LIN {X 0,Y 523.911,Z 275.225,A -85,B 0,C 180,E1 -4740.684,E2 -4740.684} C_VEL
LIN {X 0,Y 523.877,Z 275.226,A -85,B 0,C 180,E1 -4743.728,E2 -4743.728} C_VEL
LIN {X 0,Y 523.895,Z 275.245,A -85,B 0,C 180,E1 -4745.635,E2 -4745.635} C_VEL
LIN {X 0,Y 525.895,Z 284.56,A -85,B 0,C 180,E1 -4746.994,E2 -4746.994} C_VEL
LIN {X 0,Y 525.585,Z 301.308,A -85,B 0,C 180,E1 -4749.228,E2 -4749.228} C_VEL
LIN {X 0,Y 524.945,Z 326.375,A -85,B 0,C 180,E1 -4752.472,E2 -4752.472} C_VEL
LIN {X 0,Y 524.516,Z 345.364,A -85,B 0,C 180,E1 -4754.915,E2 -4754.915} C_VEL
LIN {X 0,Y 525.812,Z 356.161,A -85,B 0,C 180,E1 -4755.107,E2 -4755.107} C_VEL
LIN {X 0,Y 525.364,Z 452.042,A -85,B 0,C 180,E1 -4756.44,E2 -4756.44} C_VEL
LIN {X 0,Y 525.191,Z 462.116,A -85,B 0,C 180,E1 -4756.657,E2 -4756.657} C_VEL
LIN {X 0,Y 525.048,Z 472.823,A -85,B 0,C 180,E1 -4756.998,E2 -4756.998} C_VEL
LIN {X 0,Y 524.857,Z 483.102,A -85,B 0,C 180,E1 -4757.435,E2 -4757.435} C_VEL
LIN {X 0,Y 524.646,Z 493.466,A -85,B 0,C 180,E1 -4758.001,E2 -4758.001} C_VEL
LIN {X 0,Y 524.354,Z 503.711,A -85,B 0,C 180,E1 -4758.698,E2 -4758.698} C_VEL
LIN {X 0,Y 524.185,Z 512.016,A -85,B 0,C 180,E1 -4759.379,E2 -4759.379} C_VEL
LIN {X 0,Y 523.994,Z 520.012,A -85,B 0,C 180,E1 -4760.156,E2 -4760.156} C_VEL
LIN {X 0,Y 523.81,Z 528.29,A -85,B 0,C 180,E1 -4761.126,E2 -4761.126} C_VEL
LIN {X 0,Y 523.66,Z 535.18,A -85,B 0,C 180,E1 -4762.095,E2 -4762.095} C_VEL
LIN {X 0,Y 523.509,Z 540.935,A -85,B 0,C 180,E1 -4763.063,E2 -4763.063} C_VEL
LIN {X 0,Y 523.494,Z 546.516,A -85,B 0,C 180,E1 -4764.223,E2 -4764.223} C_VEL
LIN {X 0,Y 523.362,Z 550.893,A -85,B 0,C 180,E1 -4765.381,E2 -4765.381} C_VEL
LIN {X 0,Y 523.44,Z 553.228,A -85,B 0,C 180,E1 -4766.153,E2 -4766.153} C_VEL
LIN {X 0,Y 523.331,Z 556.518,A -85,B 0,C 180,E1 -4767.693,E2 -4767.693} C_VEL
LIN {X 0,Y 523.251,Z 558.064,A -85,B 0,C 180,E1 -4769.232,E2 -4769.232} C_VEL
LIN {X 0,Y 523.253,Z 558.357,A -85,B 0,C 180,E1 -4770.002,E2 -4770.002} C_VEL
LIN {X 0,Y 523.272,Z 557.477,A -85,B 0,C 180,E1 -4771.541,E2 -4771.541} C_VEL
LIN {X 0,Y 523.332,Z 556.501,A -85,B 0,C 180,E1 -4772.31,E2 -4772.31} C_VEL
LIN {X 0,Y 523.441,Z 553.195,A -85,B 0,C 180,E1 -4773.85,E2 -4773.85} C_VEL
LIN {X 0,Y 523.387,Z 549.529,A -85,B 0,C 180,E1 -4775.008,E2 -4775.008} C_VEL
LIN {X 0,Y 523.437,Z 544.168,A -85,B 0,C 180,E1 -4776.28,E2 -4776.28} C_VEL
LIN {X 0,Y 523.593,Z 538.647,A -85,B 0,C 180,E1 -4777.327,E2 -4777.327} C_VEL
LIN {X 0,Y 523.729,Z 532.476,A -85,B 0,C 180,E1 -4778.295,E2 -4778.295} C_VEL
LIN {X 0,Y 523.867,Z 525.025,A -85,B 0,C 180,E1 -4779.265,E2 -4779.265} C_VEL
LIN {X 0,Y 524.057,Z 515.954,A -85,B 0,C 180,E1 -4780.236,E2 -4780.236} C_VEL
LIN {X 0,Y 524.311,Z 507.212,A -85,B 0,C 180,E1 -4781.012,E2 -4781.012} C_VEL
LIN {X 0,Y 524.498,Z 498.064,A -85,B 0,C 180,E1 -4781.689,E2 -4781.689} C_VEL
LIN {X 0,Y 524.739,Z 487.826,A -85,B 0,C 180,E1 -4782.306,E2 -4782.306} C_VEL
LIN {X 0,Y 524.881,Z 478.436,A -85,B 0,C 180,E1 -4782.764,E2 -4782.764} C_VEL
LIN {X 0,Y 525.092,Z 467.337,A -85,B 0,C 180,E1 -4783.177,E2 -4783.177} C_VEL
LIN {X 0,Y 525.251,Z 456.288,A -85,B 0,C 180,E1 -4783.468,E2 -4783.468} C_VEL
LIN {X 0,Y 525.424,Z 437.769,A -85,B 0,C 180,E1 -4783.759,E2 -4783.759} C_VEL
LIN {X 0,Y 525.617,Z 353.51,A -85,B 0,C 180,E1 -4784.922,E2 -4784.922} C_VEL
LIN {X 0,Y 524.511,Z 344.96,A -85,B 0,C 180,E1 -4785.093,E2 -4785.093} C_VEL
LIN {X 0,Y 524.909,Z 321.05,A -85,B 0,C 180,E1 -4788.082,E2 -4788.082} C_VEL
LIN {X 0,Y 525.419,Z 296.571,A -85,B 0,C 180,E1 -4791.17,E2 -4791.17} C_VEL
LIN {X 0,Y 525.489,Z 283.518,A -85,B 0,C 180,E1 -4792.82,E2 -4792.82} C_VEL
LIN {X 0,Y 523.903,Z 275.226,A -85,B 0,C 180,E1 -4793.939,E2 -4793.939} C_VEL
LIN {X 0,Y 523.886,Z 275.232,A -85,B 0,C 180,E1 -4797.135,E2 -4797.135} C_VEL
LIN {X 0,Y 523.886,Z 275.23,A -85,B 0,C 180,E1 -4799.758,E2 -4799.758} C_VEL
LIN {X 0,Y 523.923,Z 275.219,A -85,B 0,C 180,E1 -4802.448,E2 -4802.448} C_VEL
LIN {X 0,Y 523.912,Z 275.225,A -85,B 0,C 180,E1 -4805.225,E2 -4805.225} C_VEL
LIN {X 0,Y 523.903,Z 275.225,A -85,B 0,C 180,E1 -4808.1,E2 -4808.1} C_VEL
LIN {X 0,Y 523.946,Z 275.22,A -85,B 0,C 180,E1 -4811.31,E2 -4811.31} C_VEL
LIN {X 0,Y 523.938,Z 275.217,A -85,B 0,C 180,E1 -4814.69,E2 -4814.69} C_VEL
LIN {X 0,Y 523.937,Z 275.224,A -85,B 0,C 180,E1 -4817.88,E2 -4817.88} C_VEL
LIN {X 0,Y 523.958,Z 275.221,A -85,B 0,C 180,E1 -4819.922,E2 -4819.922} C_VEL
LIN {X 0,Y 523.899,Z 275.22,A -85,B 0,C 180,E1 -4822.868,E2 -4822.868} C_VEL
LIN {X 0,Y 523.923,Z 275.218,A -85,B 0,C 180,E1 -4825.709,E2 -4825.709} C_VEL
LIN {X 0,Y 523.908,Z 275.224,A -85,B 0,C 180,E1 -4828.455,E2 -4828.455} C_VEL
LIN {X 0,Y 523.924,Z 275.216,A -85,B 0,C 180,E1 -4831.125,E2 -4831.125} C_VEL
LIN {X 0,Y 523.962,Z 275.215,A -85,B 0,C 180,E1 -4833.977,E2 -4833.977} C_VEL
LIN {X 0,Y 523.942,Z 275.222,A -85,B 0,C 180,E1 -4836.271,E2 -4836.271} C_VEL
LIN {X 0,Y 523.93,Z 275.224,A -85,B 0,C 180,E1 -4838.766,E2 -4838.766} C_VEL
LIN {X 0,Y 523.922,Z 275.22,A -85,B 0,C 180,E1 -4841.22,E2 -4841.22} C_VEL
LIN {X 0,Y 523.912,Z 275.22,A -85,B 0,C 180,E1 -4843.639,E2 -4843.639} C_VEL
LIN {X 0,Y 523.921,Z 275.219,A -85,B 0,C 180,E1 -4846.028,E2 -4846.028} C_VEL
LIN {X 0,Y 523.986,Z 275.217,A -85,B 0,C 180,E1 -4849.177,E2 -4849.177} C_VEL
LIN {X 0,Y 523.993,Z 275.213,A -85,B 0,C 180,E1 -4852.292,E2 -4852.292} C_VEL
LIN {X 0,Y 524.063,Z 275.207,A -85,B 0,C 180,E1 -4854.614,E2 -4854.614} C_VEL
LIN {X 0,Y 524.333,Z 275.177,A -85,B 0,C 180,E1 -4858.848,E2 -4858.848} C_VEL
LIN {X 0,Y 524.182,Z 275.432,A -85,B 0,C 180,E1 -4859.136,E2 -4859.136} C_VEL
LIN {X 0,Y 524.103,Z 293.691,A -85,B 0,C 180,E1 -4861.537,E2 -4861.537} C_VEL
LIN {X 0,Y 523.968,Z 312.922,A -85,B 0,C 180,E1 -4864.231,E2 -4864.231} C_VEL
LIN {X 0,Y 523.96,Z 332.201,A -85,B 0,C 180,E1 -4867.108,E2 -4867.108} C_VEL
LIN {X 0,Y 523.901,Z 338.208,A -85,B 0,C 180,E1 -4868.029,E2 -4868.029} C_VEL
LIN {X 0,Y 525.089,Z 347.219,A -85,B 0,C 180,E1 -4868.196,E2 -4868.196} C_VEL
LIN {X 0,Y 524.765,Z 417.596,A -85,B 0,C 180,E1 -4869.224,E2 -4869.224} C_VEL
LIN {X 0,Y 524.66,Z 428.807,A -85,B 0,C 180,E1 -4869.518,E2 -4869.518} C_VEL
LIN {X 0,Y 524.486,Z 439.253,A -85,B 0,C 180,E1 -4869.935,E2 -4869.935} C_VEL
LIN {X 0,Y 524.371,Z 448.273,A -85,B 0,C 180,E1 -4870.425,E2 -4870.425} C_VEL
LIN {X 0,Y 524.149,Z 456.892,A -85,B 0,C 180,E1 -4871.016,E2 -4871.016} C_VEL
LIN {X 0,Y 524.006,Z 463.952,A -85,B 0,C 180,E1 -4871.606,E2 -4871.606} C_VEL
LIN {X 0,Y 523.848,Z 471.672,A -85,B 0,C 180,E1 -4872.396,E2 -4872.396} C_VEL
LIN {X 0,Y 523.691,Z 478.027,A -85,B 0,C 180,E1 -4873.188,E2 -4873.188} C_VEL
LIN {X 0,Y 523.626,Z 483.278,A -85,B 0,C 180,E1 -4873.981,E2 -4873.981} C_VEL
LIN {X 0,Y 523.509,Z 488.105,A -85,B 0,C 180,E1 -4874.869,E2 -4874.869} C_VEL
LIN {X 0,Y 523.456,Z 492.829,A -85,B 0,C 180,E1 -4875.977,E2 -4875.977} C_VEL
LIN {X 0,Y 523.363,Z 496.529,A -85,B 0,C 180,E1 -4877.184,E2 -4877.184} C_VEL
LIN {X 0,Y 523.312,Z 498.218,A -85,B 0,C 180,E1 -4877.993,E2 -4877.993} C_VEL
LIN {X 0,Y 523.273,Z 499.294,A -85,B 0,C 180,E1 -4878.805,E2 -4878.805} C_VEL
LIN {X 0,Y 523.3,Z 499.96,A -85,B 0,C 180,E1 -4879.941,E2 -4879.941} C_VEL
LIN {X 0,Y 523.293,Z 499.303,A -85,B 0,C 180,E1 -4881.262,E2 -4881.262} C_VEL
LIN {X 0,Y 523.338,Z 498.18,A -85,B 0,C 180,E1 -4882.097,E2 -4882.097} C_VEL
LIN {X 0,Y 523.434,Z 495.273,A -85,B 0,C 180,E1 -4883.334,E2 -4883.334} C_VEL
LIN {X 0,Y 523.442,Z 492.023,A -85,B 0,C 180,E1 -4884.304,E2 -4884.304} C_VEL
LIN {X 0,Y 523.539,Z 486.934,A -85,B 0,C 180,E1 -4885.441,E2 -4885.441} C_VEL
LIN {X 0,Y 523.669,Z 480.771,A -85,B 0,C 180,E1 -4886.503,E2 -4886.503} C_VEL
LIN {X 0,Y 523.776,Z 473.401,A -85,B 0,C 180,E1 -4887.483,E2 -4887.483} C_VEL
LIN {X 0,Y 523.923,Z 466.588,A -85,B 0,C 180,E1 -4888.22,E2 -4888.22} C_VEL
LIN {X 0,Y 524.121,Z 458.342,A -85,B 0,C 180,E1 -4888.947,E2 -4888.947} C_VEL
LIN {X 0,Y 524.3,Z 450.697,A -85,B 0,C 180,E1 -4889.496,E2 -4889.496} C_VEL
LIN {X 0,Y 524.446,Z 441.98,A -85,B 0,C 180,E1 -4890.002,E2 -4890.002} C_VEL
LIN {X 0,Y 524.601,Z 432.241,A -85,B 0,C 180,E1 -4890.436,E2 -4890.436} C_VEL
LIN {X 0,Y 524.675,Z 423.214,A -85,B 0,C 180,E1 -4890.728,E2 -4890.728} C_VEL
LIN {X 0,Y 524.225,Z 417.513,A -85,B 0,C 180,E1 -4890.884,E2 -4890.884} C_VEL
LIN {X 0,Y 521.507,Z 408.208,A -85,B 0,C 180,E1 -4891.109,E2 -4891.109} C_VEL
LIN {X 0,Y 518.637,Z 398.829,A -85,B 0,C 180,E1 -4891.294,E2 -4891.294} C_VEL
LIN {X 0,Y 517.958,Z 393.003,A -85,B 0,C 180,E1 -4891.388,E2 -4891.388} C_VEL
LIN {X 0,Y 518.044,Z 346.377,A -85,B 0,C 180,E1 -4892.063,E2 -4892.063} C_VEL
LIN {X 0,Y 516.884,Z 338.57,A -85,B 0,C 180,E1 -4892.229,E2 -4892.229} C_VEL
LIN {X 0,Y 517.133,Z 323.91,A -85,B 0,C 180,E1 -4894.806,E2 -4894.806} C_VEL
LIN {X 0,Y 517.415,Z 308.728,A -85,B 0,C 180,E1 -4897.433,E2 -4897.433} C_VEL
LIN {X 0,Y 517.746,Z 293.76,A -85,B 0,C 180,E1 -4900.088,E2 -4900.088} C_VEL
LIN {X 0,Y 517.911,Z 282.047,A -85,B 0,C 180,E1 -4902.199,E2 -4902.199} C_VEL
LIN {X 0,Y 516.885,Z 276.103,A -85,B 0,C 180,E1 -4903.332,E2 -4903.332} C_VEL
LIN {X 0,Y 516.87,Z 276.097,A -85,B 0,C 180,E1 -4906.109,E2 -4906.109} C_VEL
LIN {X 0,Y 516.904,Z 276.091,A -85,B 0,C 180,E1 -4908.401,E2 -4908.401} C_VEL
LIN {X 0,Y 516.865,Z 276.102,A -85,B 0,C 180,E1 -4911.285,E2 -4911.285} C_VEL
LIN {X 0,Y 516.854,Z 276.097,A -85,B 0,C 180,E1 -4914.673,E2 -4914.673} C_VEL
LIN {X 0,Y 516.889,Z 276.096,A -85,B 0,C 180,E1 -4917.459,E2 -4917.459} C_VEL
LIN {X 0,Y 516.9,Z 276.092,A -85,B 0,C 180,E1 -4920.696,E2 -4920.696} C_VEL
LIN {X 0,Y 516.88,Z 276.097,A -85,B 0,C 180,E1 -4923.819,E2 -4923.819} C_VEL
LIN {X 0,Y 516.842,Z 276.103,A -85,B 0,C 180,E1 -4926.776,E2 -4926.776} C_VEL
LIN {X 0,Y 516.909,Z 276.09,A -85,B 0,C 180,E1 -4929.742,E2 -4929.742} C_VEL
LIN {X 0,Y 516.896,Z 276.1,A -85,B 0,C 180,E1 -4932.595,E2 -4932.595} C_VEL
LIN {X 0,Y 516.935,Z 276.095,A -85,B 0,C 180,E1 -4935.03,E2 -4935.03} C_VEL
LIN {X 0,Y 516.972,Z 276.082,A -85,B 0,C 180,E1 -4938.233,E2 -4938.233} C_VEL
LIN {X 0,Y 516.923,Z 276.096,A -85,B 0,C 180,E1 -4941.398,E2 -4941.398} C_VEL
LIN {X 0,Y 516.986,Z 276.08,A -85,B 0,C 180,E1 -4944.538,E2 -4944.538} C_VEL
LIN {X 0,Y 517.074,Z 276.079,A -85,B 0,C 180,E1 -4947.662,E2 -4947.662} C_VEL
LIN {X 0,Y 517.068,Z 276.076,A -85,B 0,C 180,E1 -4949.998,E2 -4949.998} C_VEL
LIN {X 0,Y 517.074,Z 276.072,A -85,B 0,C 180,E1 -4952.335,E2 -4952.335} C_VEL
LIN {X 0,Y 516.971,Z 276.09,A -85,B 0,C 180,E1 -4956.241,E2 -4956.241} C_VEL
LIN {X 0,Y 516.907,Z 276.09,A -85,B 0,C 180,E1 -4959.388,E2 -4959.388} C_VEL
LIN {X 0,Y 516.952,Z 276.086,A -85,B 0,C 180,E1 -4961.804,E2 -4961.804} C_VEL
LIN {X 0,Y 516.934,Z 276.089,A -85,B 0,C 180,E1 -4965.14,E2 -4965.14} C_VEL
LIN {X 0,Y 516.905,Z 276.092,A -85,B 0,C 180,E1 -4968.219,E2 -4968.219} C_VEL
LIN {X 0,Y 516.893,Z 276.098,A -85,B 0,C 180,E1 -4970.698,E2 -4970.698} C_VEL
LIN {X 0,Y 516.845,Z 276.106,A -85,B 0,C 180,E1 -4973.221,E2 -4973.221} C_VEL
LIN {X 0,Y 516.873,Z 276.094,A -85,B 0,C 180,E1 -4976.179,E2 -4976.179} C_VEL
LIN {X 0,Y 516.904,Z 276.099,A -85,B 0,C 180,E1 -4979.301,E2 -4979.301} C_VEL
LIN {X 0,Y 516.876,Z 276.094,A -85,B 0,C 180,E1 -4982.539,E2 -4982.539} C_VEL
LIN {X 0,Y 516.846,Z 276.101,A -85,B 0,C 180,E1 -4985.326,E2 -4985.326} C_VEL
LIN {X 0,Y 516.854,Z 276.107,A -85,B 0,C 180,E1 -4987.939,E2 -4987.939} C_VEL
LIN {X 0,Y 516.855,Z 276.098,A -85,B 0,C 180,E1 -4990.737,E2 -4990.737} C_VEL
LIN {X 0,Y 516.852,Z 276.098,A -85,B 0,C 180,E1 -4992.827,E2 -4992.827} C_VEL
LIN {X 0,Y 516.862,Z 276.097,A -85,B 0,C 180,E1 -4995.003,E2 -4995.003} C_VEL
LIN {X 0,Y 516.88,Z 276.102,A -85,B 0,C 180,E1 -4998.394,E2 -4998.394} C_VEL
LIN {X 0,Y 516.841,Z 276.1,A -85,B 0,C 180,E1 -5001.28,E2 -5001.28} C_VEL
LIN {X 0,Y 516.845,Z 276.099,A -85,B 0,C 180,E1 -5004.217,E2 -5004.217} C_VEL
LIN {X 0,Y 516.835,Z 276.109,A -85,B 0,C 180,E1 -5007.048,E2 -5007.048} C_VEL
LIN {X 0,Y 516.854,Z 276.098,A -85,B 0,C 180,E1 -5009.793,E2 -5009.793} C_VEL
LIN {X 0,Y 516.88,Z 276.094,A -85,B 0,C 180,E1 -5012.464,E2 -5012.464} C_VEL
LIN {X 0,Y 516.861,Z 276.1,A -85,B 0,C 180,E1 -5015.069,E2 -5015.069} C_VEL
LIN {X 0,Y 516.859,Z 276.107,A -85,B 0,C 180,E1 -5017.621,E2 -5017.621} C_VEL
LIN {X 0,Y 516.875,Z 276.098,A -85,B 0,C 180,E1 -5020.127,E2 -5020.127} C_VEL
LIN {X 0,Y 516.873,Z 276.095,A -85,B 0,C 180,E1 -5022.594,E2 -5022.594} C_VEL
LIN {X 0,Y 516.891,Z 276.092,A -85,B 0,C 180,E1 -5025.028,E2 -5025.028} C_VEL
LIN {X 0,Y 516.944,Z 276.096,A -85,B 0,C 180,E1 -5028.233,E2 -5028.233} C_VEL
LIN {X 0,Y 516.912,Z 276.089,A -85,B 0,C 180,E1 -5031.398,E2 -5031.398} C_VEL
LIN {X 0,Y 517.005,Z 276.088,A -85,B 0,C 180,E1 -5034.539,E2 -5034.539} C_VEL
LIN {X 0,Y 517.019,Z 276.076,A -85,B 0,C 180,E1 -5037.662,E2 -5037.662} C_VEL
LIN {X 0,Y 517.036,Z 276.082,A -85,B 0,C 180,E1 -5040.778,E2 -5040.778} C_VEL
LIN {X 0,Y 516.986,Z 276.09,A -85,B 0,C 180,E1 -5043.117,E2 -5043.117} C_VEL
LIN {X 0,Y 516.952,Z 276.085,A -85,B 0,C 180,E1 -5046.243,E2 -5046.243} C_VEL
LIN {X 0,Y 516.895,Z 276.102,A -85,B 0,C 180,E1 -5049.39,E2 -5049.39} C_VEL
LIN {X 0,Y 516.921,Z 276.094,A -85,B 0,C 180,E1 -5051.825,E2 -5051.825} C_VEL
LIN {X 0,Y 516.885,Z 276.094,A -85,B 0,C 180,E1 -5055.149,E2 -5055.149} C_VEL
LIN {X 0,Y 516.865,Z 276.101,A -85,B 0,C 180,E1 -5058.224,E2 -5058.224} C_VEL
LIN {X 0,Y 516.857,Z 276.098,A -85,B 0,C 180,E1 -5060.703,E2 -5060.703} C_VEL
LIN {X 0,Y 516.838,Z 276.099,A -85,B 0,C 180,E1 -5063.225,E2 -5063.225} C_VEL
LIN {X 0,Y 516.889,Z 276.099,A -85,B 0,C 180,E1 -5066.199,E2 -5066.199} C_VEL
LIN {X 0,Y 516.869,Z 276.096,A -85,B 0,C 180,E1 -5069.307,E2 -5069.307} C_VEL
LIN {X 0,Y 516.844,Z 276.105,A -85,B 0,C 180,E1 -5072.546,E2 -5072.546} C_VEL
LIN {X 0,Y 516.833,Z 276.103,A -85,B 0,C 180,E1 -5075.335,E2 -5075.335} C_VEL
LIN {X 0,Y 516.834,Z 276.099,A -85,B 0,C 180,E1 -5077.946,E2 -5077.946} C_VEL
LIN {X 0,Y 516.838,Z 276.102,A -85,B 0,C 180,E1 -5080.745,E2 -5080.745} C_VEL
LIN {X 0,Y 516.842,Z 276.101,A -85,B 0,C 180,E1 -5083.907,E2 -5083.907} C_VEL
LIN {X 0,Y 516.844,Z 276.1,A -85,B 0,C 180,E1 -5086.111,E2 -5086.111} C_VEL
LIN {X 0,Y 516.879,Z 276.094,A -85,B 0,C 180,E1 -5088.402,E2 -5088.402} C_VEL
LIN {X 0,Y 516.841,Z 276.101,A -85,B 0,C 180,E1 -5091.287,E2 -5091.287} C_VEL
LIN {X 0,Y 516.83,Z 276.101,A -85,B 0,C 180,E1 -5094.675,E2 -5094.675} C_VEL
LIN {X 0,Y 516.864,Z 276.096,A -85,B 0,C 180,E1 -5097.462,E2 -5097.462} C_VEL
LIN {X 0,Y 516.879,Z 276.101,A -85,B 0,C 180,E1 -5100.698,E2 -5100.698} C_VEL
LIN {X 0,Y 516.858,Z 276.101,A -85,B 0,C 180,E1 -5103.822,E2 -5103.822} C_VEL
LIN {X 0,Y 516.87,Z 276.261,A -85,B 0,C 180,E1 -5105.441,E2 -5105.441} C_VEL
LIN {X 0,Y 519.105,Z 286.956,A -85,B 0,C 180,E1 -5107.018,E2 -5107.018} C_VEL
LIN {X 0,Y 518.465,Z 309.085,A -85,B 0,C 180,E1 -5109.988,E2 -5109.988} C_VEL
LIN {X 0,Y 517.848,Z 332.375,A -85,B 0,C 180,E1 -5113.038,E2 -5113.038} C_VEL
LIN {X 0,Y 517.537,Z 345.311,A -85,B 0,C 180,E1 -5114.727,E2 -5114.727} C_VEL
LIN {X 0,Y 518.937,Z 357.146,A -85,B 0,C 180,E1 -5114.94,E2 -5114.94} C_VEL
LIN {X 0,Y 518.411,Z 451.86,A -85,B 0,C 180,E1 -5116.279,E2 -5116.279} C_VEL
LIN {X 0,Y 518.229,Z 461.905,A -85,B 0,C 180,E1 -5116.499,E2 -5116.499} C_VEL
LIN {X 0,Y 518.084,Z 471.985,A -85,B 0,C 180,E1 -5116.82,E2 -5116.82} C_VEL
LIN {X 0,Y 517.906,Z 482.391,A -85,B 0,C 180,E1 -5117.264,E2 -5117.264} C_VEL
LIN {X 0,Y 517.674,Z 492.508,A -85,B 0,C 180,E1 -5117.815,E2 -5117.815} C_VEL
LIN {X 0,Y 517.342,Z 503.137,A -85,B 0,C 180,E1 -5118.543,E2 -5118.543} C_VEL
LIN {X 0,Y 517.174,Z 511.487,A -85,B 0,C 180,E1 -5119.234,E2 -5119.234} C_VEL
LIN {X 0,Y 516.963,Z 519.515,A -85,B 0,C 180,E1 -5120.021,E2 -5120.021} C_VEL
LIN {X 0,Y 516.743,Z 527.819,A -85,B 0,C 180,E1 -5121.004,E2 -5121.004} C_VEL
LIN {X 0,Y 516.582,Z 534.73,A -85,B 0,C 180,E1 -5121.986,E2 -5121.986} C_VEL
LIN {X 0,Y 516.433,Z 540.504,A -85,B 0,C 180,E1 -5122.967,E2 -5122.967} C_VEL
LIN {X 0,Y 516.406,Z 546.097,A -85,B 0,C 180,E1 -5124.144,E2 -5124.144} C_VEL
LIN {X 0,Y 516.272,Z 550.486,A -85,B 0,C 180,E1 -5125.317,E2 -5125.317} C_VEL
LIN {X 0,Y 516.367,Z 552.823,A -85,B 0,C 180,E1 -5126.1,E2 -5126.1} C_VEL
LIN {X 0,Y 516.257,Z 556.125,A -85,B 0,C 180,E1 -5127.661,E2 -5127.661} C_VEL
LIN {X 0,Y 516.162,Z 557.672,A -85,B 0,C 180,E1 -5129.221,E2 -5129.221} C_VEL
LIN {X 0,Y 516.164,Z 557.963,A -85,B 0,C 180,E1 -5130.002,E2 -5130.002} C_VEL
LIN {X 0,Y 516.189,Z 557.077,A -85,B 0,C 180,E1 -5131.562,E2 -5131.562} C_VEL
LIN {X 0,Y 516.258,Z 556.097,A -85,B 0,C 180,E1 -5132.342,E2 -5132.342} C_VEL
LIN {X 0,Y 516.37,Z 552.773,A -85,B 0,C 180,E1 -5133.903,E2 -5133.903} C_VEL
LIN {X 0,Y 516.315,Z 549.091,A -85,B 0,C 180,E1 -5135.077,E2 -5135.077} C_VEL
LIN {X 0,Y 516.355,Z 544.271,A -85,B 0,C 180,E1 -5136.252,E2 -5136.252} C_VEL
LIN {X 0,Y 516.501,Z 538.163,A -85,B 0,C 180,E1 -5137.428,E2 -5137.428} C_VEL
LIN {X 0,Y 516.649,Z 531.964,A -85,B 0,C 180,E1 -5138.409,E2 -5138.409} C_VEL
LIN {X 0,Y 516.816,Z 524.479,A -85,B 0,C 180,E1 -5139.392,E2 -5139.392} C_VEL
LIN {X 0,Y 517.033,Z 515.366,A -85,B 0,C 180,E1 -5140.377,E2 -5140.377} C_VEL
LIN {X 0,Y 517.281,Z 506.568,A -85,B 0,C 180,E1 -5141.164,E2 -5141.164} C_VEL
LIN {X 0,Y 517.497,Z 497.202,A -85,B 0,C 180,E1 -5141.859,E2 -5141.859} C_VEL
LIN {X 0,Y 517.746,Z 487.225,A -85,B 0,C 180,E1 -5142.464,E2 -5142.464} C_VEL
LIN {X 0,Y 517.937,Z 477.478,A -85,B 0,C 180,E1 -5142.938,E2 -5142.938} C_VEL
LIN {X 0,Y 518.136,Z 466.968,A -85,B 0,C 180,E1 -5143.332,E2 -5143.332} C_VEL
LIN {X 0,Y 518.304,Z 455.872,A -85,B 0,C 180,E1 -5143.627,E2 -5143.627} C_VEL
LIN {X 0,Y 518.489,Z 437.301,A -85,B 0,C 180,E1 -5143.922,E2 -5143.922} C_VEL
LIN {X 0,Y 518.776,Z 354.539,A -85,B 0,C 180,E1 -5145.084,E2 -5145.084} C_VEL
LIN {X 0,Y 517.523,Z 344.937,A -85,B 0,C 180,E1 -5145.272,E2 -5145.272} C_VEL
LIN {X 0,Y 518.024,Z 319.066,A -85,B 0,C 180,E1 -5148.55,E2 -5148.55} C_VEL
LIN {X 0,Y 518.448,Z 296.117,A -85,B 0,C 180,E1 -5151.469,E2 -5151.469} C_VEL
LIN {X 0,Y 518.53,Z 284.678,A -85,B 0,C 180,E1 -5152.935,E2 -5152.935} C_VEL
LIN {X 0,Y 516.88,Z 276.101,A -85,B 0,C 180,E1 -5154.122,E2 -5154.122} C_VEL
LIN {X 0,Y 516.829,Z 276.106,A -85,B 0,C 180,E1 -5156.662,E2 -5156.662} C_VEL
LIN {X 0,Y 516.877,Z 276.106,A -85,B 0,C 180,E1 -5159.518,E2 -5159.518} C_VEL
LIN {X 0,Y 516.885,Z 276.096,A -85,B 0,C 180,E1 -5162.542,E2 -5162.542} C_VEL
LIN {X 0,Y 516.859,Z 276.105,A -85,B 0,C 180,E1 -5165.329,E2 -5165.329} C_VEL
LIN {X 0,Y 516.868,Z 276.104,A -85,B 0,C 180,E1 -5167.942,E2 -5167.942} C_VEL
LIN {X 0,Y 516.871,Z 276.098,A -85,B 0,C 180,E1 -5170.74,E2 -5170.74} C_VEL
LIN {X 0,Y 516.889,Z 276.096,A -85,B 0,C 180,E1 -5172.828,E2 -5172.828} C_VEL
LIN {X 0,Y 516.905,Z 276.093,A -85,B 0,C 180,E1 -5175.009,E2 -5175.009} C_VEL
LIN {X 0,Y 516.903,Z 276.096,A -85,B 0,C 180,E1 -5178.396,E2 -5178.396} C_VEL
LIN {X 0,Y 516.866,Z 276.097,A -85,B 0,C 180,E1 -5181.283,E2 -5181.283} C_VEL
LIN {X 0,Y 516.872,Z 276.101,A -85,B 0,C 180,E1 -5184.22,E2 -5184.22} C_VEL
LIN {X 0,Y 516.873,Z 276.092,A -85,B 0,C 180,E1 -5187.052,E2 -5187.052} C_VEL
LIN {X 0,Y 516.875,Z 276.095,A -85,B 0,C 180,E1 -5189.796,E2 -5189.796} C_VEL
LIN {X 0,Y 516.903,Z 276.099,A -85,B 0,C 180,E1 -5192.466,E2 -5192.466} C_VEL
LIN {X 0,Y 516.914,Z 276.092,A -85,B 0,C 180,E1 -5195.072,E2 -5195.072} C_VEL
LIN {X 0,Y 516.882,Z 276.095,A -85,B 0,C 180,E1 -5197.623,E2 -5197.623} C_VEL
LIN {X 0,Y 516.9,Z 276.096,A -85,B 0,C 180,E1 -5200.129,E2 -5200.129} C_VEL
LIN {X 0,Y 516.899,Z 276.101,A -85,B 0,C 180,E1 -5202.596,E2 -5202.596} C_VEL
LIN {X 0,Y 516.931,Z 276.095,A -85,B 0,C 180,E1 -5205.03,E2 -5205.03} C_VEL
LIN {X 0,Y 516.97,Z 276.086,A -85,B 0,C 180,E1 -5208.234,E2 -5208.234} C_VEL
LIN {X 0,Y 516.938,Z 276.094,A -85,B 0,C 180,E1 -5211.4,E2 -5211.4} C_VEL
LIN {X 0,Y 517.007,Z 276.086,A -85,B 0,C 180,E1 -5214.54,E2 -5214.54} C_VEL
LIN {X 0,Y 517.287,Z 276.055,A -85,B 0,C 180,E1 -5218.833,E2 -5218.833} C_VEL
LIN {X 0,Y 517.153,Z 276.157,A -85,B 0,C 180,E1 -5219.1,E2 -5219.1} C_VEL
LIN {X 0,Y 517.018,Z 296.231,A -85,B 0,C 180,E1 -5221.753,E2 -5221.753} C_VEL
LIN {X 0,Y 516.944,Z 315.667,A -85,B 0,C 180,E1 -5224.484,E2 -5224.484} C_VEL
LIN {X 0,Y 516.887,Z 336.71,A -85,B 0,C 180,E1 -5227.618,E2 -5227.618} C_VEL
LIN {X 0,Y 516.913,Z 338.394,A -85,B 0,C 180,E1 -5227.844,E2 -5227.844} C_VEL
LIN {X 0,Y 518.231,Z 348.399,A -85,B 0,C 180,E1 -5228.031,E2 -5228.031} C_VEL
LIN {X 0,Y 517.818,Z 416.922,A -85,B 0,C 180,E1 -5229.054,E2 -5229.054} C_VEL
LIN {X 0,Y 517.69,Z 426.025,A -85,B 0,C 180,E1 -5229.278,E2 -5229.278} C_VEL
LIN {X 0,Y 517.57,Z 435.642,A -85,B 0,C 180,E1 -5229.625,E2 -5229.625} C_VEL
LIN {X 0,Y 517.458,Z 444.801,A -85,B 0,C 180,E1 -5230.071,E2 -5230.071} C_VEL
LIN {X 0,Y 517.205,Z 455.7,A -85,B 0,C 180,E1 -5230.769,E2 -5230.769} C_VEL
LIN {X 0,Y 517.001,Z 464.533,A -85,B 0,C 180,E1 -5231.512,E2 -5231.512} C_VEL
LIN {X 0,Y 516.848,Z 470.965,A -85,B 0,C 180,E1 -5232.167,E2 -5232.167} C_VEL
LIN {X 0,Y 516.686,Z 477.502,A -85,B 0,C 180,E1 -5232.97,E2 -5232.97} C_VEL
LIN {X 0,Y 516.588,Z 482.917,A -85,B 0,C 180,E1 -5233.774,E2 -5233.774} C_VEL
LIN {X 0,Y 516.489,Z 487.351,A -85,B 0,C 180,E1 -5234.564,E2 -5234.564} C_VEL
LIN {X 0,Y 516.382,Z 492.738,A -85,B 0,C 180,E1 -5235.796,E2 -5235.796} C_VEL
LIN {X 0,Y 516.311,Z 496.614,A -85,B 0,C 180,E1 -5237.018,E2 -5237.018} C_VEL
LIN {X 0,Y 516.215,Z 499.036,A -85,B 0,C 180,E1 -5238.249,E2 -5238.249} C_VEL
LIN {X 0,Y 516.184,Z 500.001,A -85,B 0,C 180,E1 -5239.073,E2 -5239.073} C_VEL
LIN {X 0,Y 516.218,Z 500.373,A -85,B 0,C 180,E1 -5240.061,E2 -5240.061} C_VEL
LIN {X 0,Y 516.203,Z 500.11,A -85,B 0,C 180,E1 -5240.732,E2 -5240.732} C_VEL
LIN {X 0,Y 516.24,Z 499.333,A -85,B 0,C 180,E1 -5241.566,E2 -5241.566} C_VEL
LIN {X 0,Y 516.254,Z 497.987,A -85,B 0,C 180,E1 -5242.407,E2 -5242.407} C_VEL
LIN {X 0,Y 516.378,Z 494.774,A -85,B 0,C 180,E1 -5243.672,E2 -5243.672} C_VEL
LIN {X 0,Y 516.416,Z 490.018,A -85,B 0,C 180,E1 -5244.954,E2 -5244.954} C_VEL
LIN {X 0,Y 516.569,Z 483.958,A -85,B 0,C 180,E1 -5246.12,E2 -5246.12} C_VEL
LIN {X 0,Y 516.64,Z 478.996,A -85,B 0,C 180,E1 -5246.892,E2 -5246.892} C_VEL
LIN {X 0,Y 516.801,Z 472.553,A -85,B 0,C 180,E1 -5247.719,E2 -5247.719} C_VEL
LIN {X 0,Y 516.891,Z 466.013,A -85,B 0,C 180,E1 -5248.417,E2 -5248.417} C_VEL
LIN {X 0,Y 517.124,Z 458.625,A -85,B 0,C 180,E1 -5249.069,E2 -5249.069} C_VEL
LIN {X 0,Y 517.294,Z 451.298,A -85,B 0,C 180,E1 -5249.605,E2 -5249.605} C_VEL
LIN {X 0,Y 517.439,Z 443.237,A -85,B 0,C 180,E1 -5250.087,E2 -5250.087} C_VEL
LIN {X 0,Y 517.599,Z 434.532,A -85,B 0,C 180,E1 -5250.497,E2 -5250.497} C_VEL
LIN {X 0,Y 517.722,Z 425.076,A -85,B 0,C 180,E1 -5250.828,E2 -5250.828} C_VEL
LIN {X 0,Y 517.783,Z 414.859,A -85,B 0,C 180,E1 -5251.066,E2 -5251.066} C_VEL
LIN {X 0,Y 517.958,Z 393.003,A -85,B 0,C 180,E1 -5251.388,E2 -5251.388} C_VEL
LIN {X 0,Y 517.306,Z 387.196,A -85,B 0,C 180,E1 -5251.488,E2 -5251.488} C_VEL
LIN {X 0,Y 511.788,Z 368.498,A -85,B 0,C 180,E1 -5251.898,E2 -5251.898} C_VEL
LIN {X 0,Y 511.203,Z 362.693,A -85,B 0,C 180,E1 -5252.001,E2 -5252.001} C_VEL
LIN {X 0,Y 511.161,Z 347.274,A -85,B 0,C 180,E1 -5252.232,E2 -5252.232} C_VEL
LIN {X 0,Y 509.866,Z 338.629,A -85,B 0,C 180,E1 -5252.416,E2 -5252.416} C_VEL
LIN {X 0,Y 510.138,Z 323.365,A -85,B 0,C 180,E1 -5255.112,E2 -5255.112} C_VEL
LIN {X 0,Y 510.552,Z 306.776,A -85,B 0,C 180,E1 -5258.026,E2 -5258.026} C_VEL
LIN {X 0,Y 510.866,Z 290.079,A -85,B 0,C 180,E1 -5261.039,E2 -5261.039} C_VEL
LIN {X 0,Y 510.894,Z 282.659,A -85,B 0,C 180,E1 -5262.382,E2 -5262.382} C_VEL
LIN {X 0,Y 509.841,Z 276.98,A -85,B 0,C 180,E1 -5263.495,E2 -5263.495} C_VEL
LIN {X 0,Y 509.807,Z 276.977,A -85,B 0,C 180,E1 -5266.43,E2 -5266.43} C_VEL
LIN {X 0,Y 509.829,Z 276.982,A -85,B 0,C 180,E1 -5269.304,E2 -5269.304} C_VEL
LIN {X 0,Y 509.808,Z 276.981,A -85,B 0,C 180,E1 -5271.793,E2 -5271.793} C_VEL
LIN {X 0,Y 509.818,Z 276.973,A -85,B 0,C 180,E1 -5274.623,E2 -5274.623} C_VEL
LIN {X 0,Y 509.855,Z 276.973,A -85,B 0,C 180,E1 -5277.482,E2 -5277.482} C_VEL
LIN {X 0,Y 509.85,Z 276.975,A -85,B 0,C 180,E1 -5280.276,E2 -5280.276} C_VEL
LIN {X 0,Y 509.821,Z 276.973,A -85,B 0,C 180,E1 -5282.942,E2 -5282.942} C_VEL
LIN {X 0,Y 509.834,Z 276.972,A -85,B 0,C 180,E1 -5285.573,E2 -5285.573} C_VEL
LIN {X 0,Y 509.811,Z 276.979,A -85,B 0,C 180,E1 -5288.149,E2 -5288.149} C_VEL
LIN {X 0,Y 509.847,Z 276.979,A -85,B 0,C 180,E1 -5290.681,E2 -5290.681} C_VEL
LIN {X 0,Y 509.855,Z 276.972,A -85,B 0,C 180,E1 -5293.174,E2 -5293.174} C_VEL
LIN {X 0,Y 509.847,Z 276.97,A -85,B 0,C 180,E1 -5295.633,E2 -5295.633} C_VEL
LIN {X 0,Y 509.911,Z 276.968,A -85,B 0,C 180,E1 -5298.874,E2 -5298.874} C_VEL
LIN {X 0,Y 509.879,Z 276.966,A -85,B 0,C 180,E1 -5302.077,E2 -5302.077} C_VEL
LIN {X 0,Y 509.941,Z 276.958,A -85,B 0,C 180,E1 -5304.463,E2 -5304.463} C_VEL
LIN {X 0,Y 510.042,Z 276.955,A -85,B 0,C 180,E1 -5307.629,E2 -5307.629} C_VEL
LIN {X 0,Y 510.037,Z 276.952,A -85,B 0,C 180,E1 -5309.998,E2 -5309.998} C_VEL
LIN {X 0,Y 510.043,Z 276.948,A -85,B 0,C 180,E1 -5312.367,E2 -5312.367} C_VEL
LIN {X 0,Y 509.937,Z 276.961,A -85,B 0,C 180,E1 -5315.534,E2 -5315.534} C_VEL
LIN {X 0,Y 509.875,Z 276.972,A -85,B 0,C 180,E1 -5317.92,E2 -5317.92} C_VEL
LIN {X 0,Y 509.905,Z 276.963,A -85,B 0,C 180,E1 -5321.123,E2 -5321.123} C_VEL
LIN {X 0,Y 509.844,Z 276.977,A -85,B 0,C 180,E1 -5324.363,E2 -5324.363} C_VEL
LIN {X 0,Y 509.861,Z 276.976,A -85,B 0,C 180,E1 -5326.823,E2 -5326.823} C_VEL
LIN {X 0,Y 509.9,Z 276.964,A -85,B 0,C 180,E1 -5330.152,E2 -5330.152} C_VEL
LIN {X 0,Y 509.807,Z 276.978,A -85,B 0,C 180,E1 -5333.56,E2 -5333.56} C_VEL
LIN {X 0,Y 509.825,Z 276.972,A -85,B 0,C 180,E1 -5336.358,E2 -5336.358} C_VEL
LIN {X 0,Y 509.834,Z 276.973,A -85,B 0,C 180,E1 -5338.842,E2 -5338.842} C_VEL
LIN {X 0,Y 509.801,Z 276.985,A -85,B 0,C 180,E1 -5341.586,E2 -5341.586} C_VEL
LIN {X 0,Y 509.827,Z 276.973,A -85,B 0,C 180,E1 -5344.409,E2 -5344.409} C_VEL
LIN {X 0,Y 509.792,Z 276.979,A -85,B 0,C 180,E1 -5347.337,E2 -5347.337} C_VEL
LIN {X 0,Y 509.811,Z 276.979,A -85,B 0,C 180,E1 -5350.378,E2 -5350.378} C_VEL
LIN {X 0,Y 509.792,Z 276.977,A -85,B 0,C 180,E1 -5353.058,E2 -5353.058} C_VEL
LIN {X 0,Y 509.789,Z 276.979,A -85,B 0,C 180,E1 -5355.789,E2 -5355.789} C_VEL
LIN {X 0,Y 509.822,Z 276.983,A -85,B 0,C 180,E1 -5358.57,E2 -5358.57} C_VEL
LIN {X 0,Y 509.81,Z 276.974,A -85,B 0,C 180,E1 -5361.782,E2 -5361.782} C_VEL
LIN {X 0,Y 509.8,Z 276.982,A -85,B 0,C 180,E1 -5364.619,E2 -5364.619} C_VEL
LIN {X 0,Y 509.813,Z 276.977,A -85,B 0,C 180,E1 -5367.477,E2 -5367.477} C_VEL
LIN {X 0,Y 509.835,Z 276.971,A -85,B 0,C 180,E1 -5370.265,E2 -5370.265} C_VEL
LIN {X 0,Y 509.837,Z 276.975,A -85,B 0,C 180,E1 -5372.941,E2 -5372.941} C_VEL
LIN {X 0,Y 509.822,Z 276.982,A -85,B 0,C 180,E1 -5375.571,E2 -5375.571} C_VEL
LIN {X 0,Y 509.794,Z 276.979,A -85,B 0,C 180,E1 -5378.147,E2 -5378.147} C_VEL
LIN {X 0,Y 509.808,Z 276.975,A -85,B 0,C 180,E1 -5380.679,E2 -5380.679} C_VEL
LIN {X 0,Y 509.83,Z 276.972,A -85,B 0,C 180,E1 -5383.172,E2 -5383.172} C_VEL
LIN {X 0,Y 509.818,Z 276.977,A -85,B 0,C 180,E1 -5385.632,E2 -5385.632} C_VEL
LIN {X 0,Y 509.861,Z 276.969,A -85,B 0,C 180,E1 -5388.873,E2 -5388.873} C_VEL
LIN {X 0,Y 509.891,Z 276.969,A -85,B 0,C 180,E1 -5392.077,E2 -5392.077} C_VEL
LIN {X 0,Y 509.952,Z 276.965,A -85,B 0,C 180,E1 -5394.464,E2 -5394.464} C_VEL
LIN {X 0,Y 509.992,Z 276.952,A -85,B 0,C 180,E1 -5397.63,E2 -5397.63} C_VEL
LIN {X 0,Y 509.987,Z 276.952,A -85,B 0,C 180,E1 -5400,E2 -5400} C_VEL
LIN {X 0,Y 509.927,Z 276.969,A -85,B 0,C 180,E1 -5403.16,E2 -5403.16} C_VEL
LIN {X 0,Y 509.919,Z 276.961,A -85,B 0,C 180,E1 -5406.33,E2 -5406.33} C_VEL
LIN {X 0,Y 509.857,Z 276.97,A -85,B 0,C 180,E1 -5408.721,E2 -5408.721} C_VEL
LIN {X 0,Y 509.89,Z 276.969,A -85,B 0,C 180,E1 -5411.932,E2 -5411.932} C_VEL
LIN {X 0,Y 509.833,Z 276.974,A -85,B 0,C 180,E1 -5415.243,E2 -5415.243} C_VEL
LIN {X 0,Y 509.828,Z 276.981,A -85,B 0,C 180,E1 -5418.002,E2 -5418.002} C_VEL
LIN {X 0,Y 509.801,Z 276.975,A -85,B 0,C 180,E1 -5421.003,E2 -5421.003} C_VEL
LIN {X 0,Y 509.795,Z 276.977,A -85,B 0,C 180,E1 -5423.565,E2 -5423.565} C_VEL
LIN {X 0,Y 509.858,Z 276.979,A -85,B 0,C 180,E1 -5426.381,E2 -5426.381} C_VEL
LIN {X 0,Y 509.825,Z 276.978,A -85,B 0,C 180,E1 -5428.847,E2 -5428.847} C_VEL
LIN {X 0,Y 509.767,Z 276.98,A -85,B 0,C 180,E1 -5431.593,E2 -5431.593} C_VEL
LIN {X 0,Y 509.804,Z 276.978,A -85,B 0,C 180,E1 -5434.417,E2 -5434.417} C_VEL
LIN {X 0,Y 509.772,Z 276.984,A -85,B 0,C 180,E1 -5437.344,E2 -5437.344} C_VEL
LIN {X 0,Y 509.794,Z 276.977,A -85,B 0,C 180,E1 -5440.386,E2 -5440.386} C_VEL
LIN {X 0,Y 509.764,Z 276.985,A -85,B 0,C 180,E1 -5443.063,E2 -5443.063} C_VEL
LIN {X 0,Y 509.785,Z 276.983,A -85,B 0,C 180,E1 -5445.797,E2 -5445.797} C_VEL
LIN {X 0,Y 509.821,Z 276.973,A -85,B 0,C 180,E1 -5448.578,E2 -5448.578} C_VEL
LIN {X 0,Y 509.784,Z 276.987,A -85,B 0,C 180,E1 -5451.795,E2 -5451.795} C_VEL
LIN {X 0,Y 509.794,Z 276.978,A -85,B 0,C 180,E1 -5454.625,E2 -5454.625} C_VEL
LIN {X 0,Y 509.83,Z 276.973,A -85,B 0,C 180,E1 -5457.484,E2 -5457.484} C_VEL
LIN {X 0,Y 509.829,Z 276.981,A -85,B 0,C 180,E1 -5460.279,E2 -5460.279} C_VEL
LIN {X 0,Y 509.797,Z 276.984,A -85,B 0,C 180,E1 -5462.944,E2 -5462.944} C_VEL
LIN {X 0,Y 509.812,Z 277.029,A -85,B 0,C 180,E1 -5465.206,E2 -5465.206} C_VEL
LIN {X 0,Y 512.249,Z 288.962,A -85,B 0,C 180,E1 -5466.988,E2 -5466.988} C_VEL
LIN {X 0,Y 511.527,Z 310.497,A -85,B 0,C 180,E1 -5469.915,E2 -5469.915} C_VEL
LIN {X 0,Y 510.904,Z 332.163,A -85,B 0,C 180,E1 -5472.801,E2 -5472.801} C_VEL
LIN {X 0,Y 510.587,Z 345.54,A -85,B 0,C 180,E1 -5474.541,E2 -5474.541} C_VEL
LIN {X 0,Y 512.004,Z 356.475,A -85,B 0,C 180,E1 -5474.742,E2 -5474.742} C_VEL
LIN {X 0,Y 511.463,Z 451.676,A -85,B 0,C 180,E1 -5476.114,E2 -5476.114} C_VEL
LIN {X 0,Y 511.296,Z 461.698,A -85,B 0,C 180,E1 -5476.338,E2 -5476.338} C_VEL
LIN {X 0,Y 511.119,Z 472.367,A -85,B 0,C 180,E1 -5476.687,E2 -5476.687} C_VEL
LIN {X 0,Y 510.93,Z 481.677,A -85,B 0,C 180,E1 -5477.087,E2 -5477.087} C_VEL
LIN {X 0,Y 510.652,Z 493.126,A -85,B 0,C 180,E1 -5477.728,E2 -5477.728} C_VEL
LIN {X 0,Y 510.349,Z 502.564,A -85,B 0,C 180,E1 -5478.384,E2 -5478.384} C_VEL
LIN {X 0,Y 510.099,Z 511.985,A -85,B 0,C 180,E1 -5479.183,E2 -5479.183} C_VEL
LIN {X 0,Y 509.86,Z 520.737,A -85,B 0,C 180,E1 -5480.081,E2 -5480.081} C_VEL
LIN {X 0,Y 509.69,Z 527.348,A -85,B 0,C 180,E1 -5480.879,E2 -5480.879} C_VEL
LIN {X 0,Y 509.504,Z 534.28,A -85,B 0,C 180,E1 -5481.874,E2 -5481.874} C_VEL
LIN {X 0,Y 509.384,Z 540.073,A -85,B 0,C 180,E1 -5482.869,E2 -5482.869} C_VEL
LIN {X 0,Y 509.298,Z 545.678,A -85,B 0,C 180,E1 -5484.062,E2 -5484.062} C_VEL
LIN {X 0,Y 509.189,Z 550.079,A -85,B 0,C 180,E1 -5485.252,E2 -5485.252} C_VEL
LIN {X 0,Y 509.276,Z 552.416,A -85,B 0,C 180,E1 -5486.045,E2 -5486.045} C_VEL
LIN {X 0,Y 509.186,Z 555.731,A -85,B 0,C 180,E1 -5487.629,E2 -5487.629} C_VEL
LIN {X 0,Y 509.075,Z 557.279,A -85,B 0,C 180,E1 -5489.211,E2 -5489.211} C_VEL
LIN {X 0,Y 509.076,Z 557.568,A -85,B 0,C 180,E1 -5490.002,E2 -5490.002} C_VEL
LIN {X 0,Y 509.11,Z 556.677,A -85,B 0,C 180,E1 -5491.584,E2 -5491.584} C_VEL
LIN {X 0,Y 509.186,Z 555.693,A -85,B 0,C 180,E1 -5492.374,E2 -5492.374} C_VEL
LIN {X 0,Y 509.281,Z 552.35,A -85,B 0,C 180,E1 -5493.958,E2 -5493.958} C_VEL
LIN {X 0,Y 509.247,Z 548.653,A -85,B 0,C 180,E1 -5495.148,E2 -5495.148} C_VEL
LIN {X 0,Y 509.284,Z 543.813,A -85,B 0,C 180,E1 -5496.339,E2 -5496.339} C_VEL
LIN {X 0,Y 509.414,Z 537.679,A -85,B 0,C 180,E1 -5497.532,E2 -5497.532} C_VEL
LIN {X 0,Y 509.578,Z 531.451,A -85,B 0,C 180,E1 -5498.527,E2 -5498.527} C_VEL
LIN {X 0,Y 509.746,Z 523.931,A -85,B 0,C 180,E1 -5499.524,E2 -5499.524} C_VEL
LIN {X 0,Y 509.968,Z 515.809,A -85,B 0,C 180,E1 -5500.422,E2 -5500.422} C_VEL
LIN {X 0,Y 510.238,Z 507.169,A -85,B 0,C 180,E1 -5501.219,E2 -5501.219} C_VEL
LIN {X 0,Y 510.463,Z 498.09,A -85,B 0,C 180,E1 -5501.919,E2 -5501.919} C_VEL
LIN {X 0,Y 510.722,Z 488.403,A -85,B 0,C 180,E1 -5502.532,E2 -5502.532} C_VEL
LIN {X 0,Y 510.964,Z 477.74,A -85,B 0,C 180,E1 -5503.067,E2 -5503.067} C_VEL
LIN {X 0,Y 511.191,Z 466.6,A -85,B 0,C 180,E1 -5503.491,E2 -5503.491} C_VEL
LIN {X 0,Y 511.354,Z 455.454,A -85,B 0,C 180,E1 -5503.791,E2 -5503.791} C_VEL
LIN {X 0,Y 511.558,Z 436.833,A -85,B 0,C 180,E1 -5504.089,E2 -5504.089} C_VEL
LIN {X 0,Y 511.893,Z 355.452,A -85,B 0,C 180,E1 -5505.253,E2 -5505.253} C_VEL
LIN {X 0,Y 510.52,Z 344.912,A -85,B 0,C 180,E1 -5505.457,E2 -5505.457} C_VEL
LIN {X 0,Y 511.053,Z 319.984,A -85,B 0,C 180,E1 -5508.647,E2 -5508.647} C_VEL
LIN {X 0,Y 511.504,Z 297.323,A -85,B 0,C 180,E1 -5511.564,E2 -5511.564} C_VEL
LIN {X 0,Y 511.617,Z 286.113,A -85,B 0,C 180,E1 -5513.021,E2 -5513.021} C_VEL
LIN {X 0,Y 509.83,Z 276.979,A -85,B 0,C 180,E1 -5514.319,E2 -5514.319} C_VEL
LIN {X 0,Y 509.81,Z 276.985,A -85,B 0,C 180,E1 -5517.059,E2 -5517.059} C_VEL
LIN {X 0,Y 509.843,Z 276.98,A -85,B 0,C 180,E1 -5519.751,E2 -5519.751} C_VEL
LIN {X 0,Y 509.862,Z 276.972,A -85,B 0,C 180,E1 -5522.773,E2 -5522.773} C_VEL
LIN {X 0,Y 509.818,Z 276.984,A -85,B 0,C 180,E1 -5525.578,E2 -5525.578} C_VEL
LIN {X 0,Y 509.837,Z 276.976,A -85,B 0,C 180,E1 -5528.337,E2 -5528.337} C_VEL
LIN {X 0,Y 509.844,Z 276.978,A -85,B 0,C 180,E1 -5531.424,E2 -5531.424} C_VEL
LIN {X 0,Y 509.84,Z 276.974,A -85,B 0,C 180,E1 -5534.666,E2 -5534.666} C_VEL
LIN {X 0,Y 509.842,Z 276.98,A -85,B 0,C 180,E1 -5538.101,E2 -5538.101} C_VEL
LIN {X 0,Y 509.839,Z 276.974,A -85,B 0,C 180,E1 -5540.647,E2 -5540.647} C_VEL
LIN {X 0,Y 509.817,Z 276.977,A -85,B 0,C 180,E1 -5543.647,E2 -5543.647} C_VEL
LIN {X 0,Y 509.839,Z 276.973,A -85,B 0,C 180,E1 -5546.538,E2 -5546.538} C_VEL
LIN {X 0,Y 509.824,Z 276.971,A -85,B 0,C 180,E1 -5549.333,E2 -5549.333} C_VEL
LIN {X 0,Y 509.868,Z 276.971,A -85,B 0,C 180,E1 -5552.053,E2 -5552.053} C_VEL
LIN {X 0,Y 509.87,Z 276.974,A -85,B 0,C 180,E1 -5554.704,E2 -5554.704} C_VEL
LIN {X 0,Y 509.853,Z 276.971,A -85,B 0,C 180,E1 -5557.441,E2 -5557.441} C_VEL
LIN {X 0,Y 509.885,Z 276.968,A -85,B 0,C 180,E1 -5559.844,E2 -5559.844} C_VEL
LIN {X 0,Y 509.856,Z 276.974,A -85,B 0,C 180,E1 -5563.174,E2 -5563.174} C_VEL
LIN {X 0,Y 509.851,Z 276.972,A -85,B 0,C 180,E1 -5565.634,E2 -5565.634} C_VEL
LIN {X 0,Y 509.901,Z 276.973,A -85,B 0,C 180,E1 -5568.875,E2 -5568.875} C_VEL
LIN {X 0,Y 509.917,Z 276.967,A -85,B 0,C 180,E1 -5572.078,E2 -5572.078} C_VEL
LIN {X 0,Y 509.956,Z 276.964,A -85,B 0,C 180,E1 -5574.464,E2 -5574.464} C_VEL
LIN {X 0,Y 510.241,Z 276.932,A -85,B 0,C 180,E1 -5578.817,E2 -5578.817} C_VEL
LIN {X 0,Y 510.124,Z 277.116,A -85,B 0,C 180,E1 -5579.063,E2 -5579.063} C_VEL
LIN {X 0,Y 509.984,Z 297.517,A -85,B 0,C 180,E1 -5581.777,E2 -5581.777} C_VEL
LIN {X 0,Y 509.913,Z 317.192,A -85,B 0,C 180,E1 -5584.546,E2 -5584.546} C_VEL
LIN {X 0,Y 509.871,Z 338.037,A -85,B 0,C 180,E1 -5587.636,E2 -5587.636} C_VEL
LIN {X 0,Y 511.347,Z 348.462,A -85,B 0,C 180,E1 -5587.845,E2 -5587.845} C_VEL
LIN {X 0,Y 510.877,Z 417.502,A -85,B 0,C 180,E1 -5588.904,E2 -5588.904} C_VEL
LIN {X 0,Y 510.726,Z 427.307,A -85,B 0,C 180,E1 -5589.156,E2 -5589.156} C_VEL
LIN {X 0,Y 510.598,Z 438.98,A -85,B 0,C 180,E1 -5589.608,E2 -5589.608} C_VEL
LIN {X 0,Y 510.389,Z 449.78,A -85,B 0,C 180,E1 -5590.212,E2 -5590.212} C_VEL
LIN {X 0,Y 510.154,Z 458.254,A -85,B 0,C 180,E1 -5590.819,E2 -5590.819} C_VEL
LIN {X 0,Y 509.968,Z 465.697,A -85,B 0,C 180,E1 -5591.473,E2 -5591.473} C_VEL
LIN {X 0,Y 509.829,Z 471.988,A -85,B 0,C 180,E1 -5592.136,E2 -5592.136} C_VEL
LIN {X 0,Y 509.637,Z 478.428,A -85,B 0,C 180,E1 -5592.95,E2 -5592.95} C_VEL
LIN {X 0,Y 509.524,Z 483.758,A -85,B 0,C 180,E1 -5593.765,E2 -5593.765} C_VEL
LIN {X 0,Y 509.396,Z 488.817,A -85,B 0,C 180,E1 -5594.713,E2 -5594.713} C_VEL
LIN {X 0,Y 509.322,Z 492.645,A -85,B 0,C 180,E1 -5595.61,E2 -5595.61} C_VEL
LIN {X 0,Y 509.298,Z 495.442,A -85,B 0,C 180,E1 -5596.433,E2 -5596.433} C_VEL
LIN {X 0,Y 509.169,Z 498.663,A -85,B 0,C 180,E1 -5597.762,E2 -5597.762} C_VEL
LIN {X 0,Y 509.115,Z 499.781,A -85,B 0,C 180,E1 -5598.512,E2 -5598.512} C_VEL
LIN {X 0,Y 509.117,Z 500.525,A -85,B 0,C 180,E1 -5599.348,E2 -5599.348} C_VEL
LIN {X 0,Y 509.148,Z 500.737,A -85,B 0,C 180,E1 -5600.188,E2 -5600.188} C_VEL
LIN {X 0,Y 509.143,Z 500.364,A -85,B 0,C 180,E1 -5601.033,E2 -5601.033} C_VEL
LIN {X 0,Y 509.171,Z 498.502,A -85,B 0,C 180,E1 -5602.373,E2 -5602.373} C_VEL
LIN {X 0,Y 509.253,Z 496.789,A -85,B 0,C 180,E1 -5603.162,E2 -5603.162} C_VEL
LIN {X 0,Y 509.299,Z 494.33,A -85,B 0,C 180,E1 -5603.997,E2 -5603.997} C_VEL
LIN {X 0,Y 509.351,Z 489.982,A -85,B 0,C 180,E1 -5605.106,E2 -5605.106} C_VEL
LIN {X 0,Y 509.508,Z 484.358,A -85,B 0,C 180,E1 -5606.194,E2 -5606.194} C_VEL
LIN {X 0,Y 509.633,Z 478.723,A -85,B 0,C 180,E1 -5607.071,E2 -5607.071} C_VEL
LIN {X 0,Y 509.731,Z 473.677,A -85,B 0,C 180,E1 -5607.732,E2 -5607.732} C_VEL
LIN {X 0,Y 509.887,Z 466.361,A -85,B 0,C 180,E1 -5608.529,E2 -5608.529} C_VEL
LIN {X 0,Y 510.106,Z 459.242,A -85,B 0,C 180,E1 -5609.169,E2 -5609.169} C_VEL
LIN {X 0,Y 510.313,Z 451.818,A -85,B 0,C 180,E1 -5609.722,E2 -5609.722} C_VEL
LIN {X 0,Y 510.438,Z 444.043,A -85,B 0,C 180,E1 -5610.199,E2 -5610.199} C_VEL
LIN {X 0,Y 510.627,Z 435.477,A -85,B 0,C 180,E1 -5610.614,E2 -5610.614} C_VEL
LIN {X 0,Y 510.738,Z 426.257,A -85,B 0,C 180,E1 -5610.951,E2 -5610.951} C_VEL
LIN {X 0,Y 510.838,Z 416.712,A -85,B 0,C 180,E1 -5611.189,E2 -5611.189} C_VEL
LIN {X 0,Y 511.203,Z 362.693,A -85,B 0,C 180,E1 -5612.001,E2 -5612.001} C_VEL
LIN {X 0,Y 510.587,Z 358.854,A -85,B 0,C 180,E1 -5612.076,E2 -5612.076} C_VEL
LIN {X 0,Y 507.785,Z 352.963,A -85,B 0,C 180,E1 -5612.239,E2 -5612.239} C_VEL
LIN {X 0,Y 504.657,Z 347.117,A -85,B 0,C 180,E1 -5612.413,E2 -5612.413} C_VEL
LIN {X 0,Y 503.554,Z 343.313,A -85,B 0,C 180,E1 -5612.501,E2 -5612.501} C_VEL
LIN {X 0,Y 502.866,Z 338.745,A -85,B 0,C 180,E1 -5612.598,E2 -5612.598} C_VEL
LIN {X 0,Y 503.279,Z 320.056,A -85,B 0,C 180,E1 -5615.916,E2 -5615.916} C_VEL
LIN {X 0,Y 503.645,Z 303.381,A -85,B 0,C 180,E1 -5618.899,E2 -5618.899} C_VEL
LIN {X 0,Y 504.084,Z 286.281,A -85,B 0,C 180,E1 -5622.008,E2 -5622.008} C_VEL
LIN {X 0,Y 503.265,Z 280.132,A -85,B 0,C 180,E1 -5623.179,E2 -5623.179} C_VEL
LIN {X 0,Y 502.802,Z 277.856,A -85,B 0,C 180,E1 -5623.641,E2 -5623.641} C_VEL
LIN {X 0,Y 502.76,Z 277.857,A -85,B 0,C 180,E1 -5626.771,E2 -5626.771} C_VEL
LIN {X 0,Y 502.809,Z 277.852,A -85,B 0,C 180,E1 -5629.007,E2 -5629.007} C_VEL
LIN {X 0,Y 502.757,Z 277.856,A -85,B 0,C 180,E1 -5632.045,E2 -5632.045} C_VEL
LIN {X 0,Y 502.787,Z 277.85,A -85,B 0,C 180,E1 -5635.035,E2 -5635.035} C_VEL
LIN {X 0,Y 502.778,Z 277.861,A -85,B 0,C 180,E1 -5637.917,E2 -5637.917} C_VEL
LIN {X 0,Y 502.801,Z 277.849,A -85,B 0,C 180,E1 -5640.712,E2 -5640.712} C_VEL
LIN {X 0,Y 502.774,Z 277.851,A -85,B 0,C 180,E1 -5643.461,E2 -5643.461} C_VEL
LIN {X 0,Y 502.761,Z 277.858,A -85,B 0,C 180,E1 -5646.085,E2 -5646.085} C_VEL
LIN {X 0,Y 502.833,Z 277.844,A -85,B 0,C 180,E1 -5649.464,E2 -5649.464} C_VEL
LIN {X 0,Y 502.819,Z 277.847,A -85,B 0,C 180,E1 -5652.092,E2 -5652.092} C_VEL
LIN {X 0,Y 502.828,Z 277.846,A -85,B 0,C 180,E1 -5655.429,E2 -5655.429} C_VEL
LIN {X 0,Y 502.877,Z 277.842,A -85,B 0,C 180,E1 -5658.716,E2 -5658.716} C_VEL
LIN {X 0,Y 502.851,Z 277.842,A -85,B 0,C 180,E1 -5661.965,E2 -5661.965} C_VEL
LIN {X 0,Y 502.898,Z 277.835,A -85,B 0,C 180,E1 -5664.385,E2 -5664.385} C_VEL
LIN {X 0,Y 503.01,Z 277.832,A -85,B 0,C 180,E1 -5667.596,E2 -5667.596} C_VEL
LIN {X 0,Y 503.006,Z 277.828,A -85,B 0,C 180,E1 -5669.998,E2 -5669.998} C_VEL
LIN {X 0,Y 503.01,Z 277.824,A -85,B 0,C 180,E1 -5672.4,E2 -5672.4} C_VEL
LIN {X 0,Y 502.894,Z 277.839,A -85,B 0,C 180,E1 -5675.612,E2 -5675.612} C_VEL
LIN {X 0,Y 502.847,Z 277.849,A -85,B 0,C 180,E1 -5678.032,E2 -5678.032} C_VEL
LIN {X 0,Y 502.871,Z 277.839,A -85,B 0,C 180,E1 -5681.281,E2 -5681.281} C_VEL
LIN {X 0,Y 502.825,Z 277.855,A -85,B 0,C 180,E1 -5684.568,E2 -5684.568} C_VEL
LIN {X 0,Y 502.807,Z 277.851,A -85,B 0,C 180,E1 -5687.066,E2 -5687.066} C_VEL
LIN {X 0,Y 502.805,Z 277.848,A -85,B 0,C 180,E1 -5689.597,E2 -5689.597} C_VEL
LIN {X 0,Y 502.792,Z 277.853,A -85,B 0,C 180,E1 -5692.698,E2 -5692.698} C_VEL
LIN {X 0,Y 502.769,Z 277.854,A -85,B 0,C 180,E1 -5695.675,E2 -5695.675} C_VEL
LIN {X 0,Y 502.781,Z 277.85,A -85,B 0,C 180,E1 -5698.371,E2 -5698.371} C_VEL
LIN {X 0,Y 502.776,Z 277.855,A -85,B 0,C 180,E1 -5701.139,E2 -5701.139} C_VEL
LIN {X 0,Y 502.783,Z 277.855,A -85,B 0,C 180,E1 -5703.99,E2 -5703.99} C_VEL
LIN {X 0,Y 502.754,Z 277.854,A -85,B 0,C 180,E1 -5707.173,E2 -5707.173} C_VEL
LIN {X 0,Y 502.76,Z 277.863,A -85,B 0,C 180,E1 -5710.011,E2 -5710.011} C_VEL
LIN {X 0,Y 502.774,Z 277.861,A -85,B 0,C 180,E1 -5712.195,E2 -5712.195} C_VEL
LIN {X 0,Y 502.752,Z 277.854,A -85,B 0,C 180,E1 -5715.466,E2 -5715.466} C_VEL
LIN {X 0,Y 502.784,Z 277.853,A -85,B 0,C 180,E1 -5718.93,E2 -5718.93} C_VEL
LIN {X 0,Y 502.753,Z 277.855,A -85,B 0,C 180,E1 -5722.042,E2 -5722.042} C_VEL
LIN {X 0,Y 502.761,Z 277.86,A -85,B 0,C 180,E1 -5725.031,E2 -5725.031} C_VEL
LIN {X 0,Y 502.735,Z 277.856,A -85,B 0,C 180,E1 -5727.911,E2 -5727.911} C_VEL
LIN {X 0,Y 502.794,Z 277.851,A -85,B 0,C 180,E1 -5730.71,E2 -5730.71} C_VEL
LIN {X 0,Y 502.831,Z 277.853,A -85,B 0,C 180,E1 -5733.432,E2 -5733.432} C_VEL
LIN {X 0,Y 502.748,Z 277.856,A -85,B 0,C 180,E1 -5736.084,E2 -5736.084} C_VEL
LIN {X 0,Y 502.741,Z 277.855,A -85,B 0,C 180,E1 -5738.686,E2 -5738.686} C_VEL
LIN {X 0,Y 502.788,Z 277.859,A -85,B 0,C 180,E1 -5741.876,E2 -5741.876} C_VEL
LIN {X 0,Y 502.78,Z 277.851,A -85,B 0,C 180,E1 -5744.66,E2 -5744.66} C_VEL
LIN {X 0,Y 502.866,Z 277.846,A -85,B 0,C 180,E1 -5748.011,E2 -5748.011} C_VEL
LIN {X 0,Y 502.816,Z 277.846,A -85,B 0,C 180,E1 -5751.155,E2 -5751.155} C_VEL
LIN {X 0,Y 502.87,Z 277.839,A -85,B 0,C 180,E1 -5753.58,E2 -5753.58} C_VEL
LIN {X 0,Y 502.871,Z 277.848,A -85,B 0,C 180,E1 -5756.795,E2 -5756.795} C_VEL
LIN {X 0,Y 502.976,Z 277.83,A -85,B 0,C 180,E1 -5759.199,E2 -5759.199} C_VEL
LIN {X 0,Y 502.843,Z 277.844,A -85,B 0,C 180,E1 -5761.601,E2 -5761.601} C_VEL
LIN {X 0,Y 502.869,Z 277.847,A -85,B 0,C 180,E1 -5763.204,E2 -5763.204} C_VEL
LIN {X 0,Y 502.868,Z 277.839,A -85,B 0,C 180,E1 -5766.419,E2 -5766.419} C_VEL
LIN {X 0,Y 502.815,Z 277.848,A -85,B 0,C 180,E1 -5768.844,E2 -5768.844} C_VEL
LIN {X 0,Y 502.833,Z 277.846,A -85,B 0,C 180,E1 -5772.102,E2 -5772.102} C_VEL
LIN {X 0,Y 502.788,Z 277.853,A -85,B 0,C 180,E1 -5775.401,E2 -5775.401} C_VEL
LIN {X 0,Y 502.786,Z 277.856,A -85,B 0,C 180,E1 -5778.123,E2 -5778.123} C_VEL
LIN {X 0,Y 502.741,Z 277.855,A -85,B 0,C 180,E1 -5781.313,E2 -5781.313} C_VEL
LIN {X 0,Y 502.747,Z 277.859,A -85,B 0,C 180,E1 -5783.916,E2 -5783.916} C_VEL
LIN {X 0,Y 502.81,Z 277.854,A -85,B 0,C 180,E1 -5786.569,E2 -5786.569} C_VEL
LIN {X 0,Y 502.772,Z 277.852,A -85,B 0,C 180,E1 -5789.291,E2 -5789.291} C_VEL
LIN {X 0,Y 502.731,Z 277.857,A -85,B 0,C 180,E1 -5792.088,E2 -5792.088} C_VEL
LIN {X 0,Y 502.76,Z 277.862,A -85,B 0,C 180,E1 -5794.968,E2 -5794.968} C_VEL
LIN {X 0,Y 502.748,Z 277.854,A -85,B 0,C 180,E1 -5797.958,E2 -5797.958} C_VEL
LIN {X 0,Y 502.757,Z 277.86,A -85,B 0,C 180,E1 -5801.072,E2 -5801.072} C_VEL
LIN {X 0,Y 502.739,Z 277.855,A -85,B 0,C 180,E1 -5804.344,E2 -5804.344} C_VEL
LIN {X 0,Y 502.735,Z 277.856,A -85,B 0,C 180,E1 -5806.772,E2 -5806.772} C_VEL
LIN {X 0,Y 502.785,Z 277.85,A -85,B 0,C 180,E1 -5809.009,E2 -5809.009} C_VEL
LIN {X 0,Y 502.733,Z 277.863,A -85,B 0,C 180,E1 -5812.047,E2 -5812.047} C_VEL
LIN {X 0,Y 502.762,Z 277.852,A -85,B 0,C 180,E1 -5815.037,E2 -5815.037} C_VEL
LIN {X 0,Y 502.752,Z 277.859,A -85,B 0,C 180,E1 -5817.919,E2 -5817.919} C_VEL
LIN {X 0,Y 502.779,Z 277.858,A -85,B 0,C 180,E1 -5820.714,E2 -5820.714} C_VEL
LIN {X 0,Y 502.753,Z 277.858,A -85,B 0,C 180,E1 -5823.464,E2 -5823.464} C_VEL
LIN {X 0,Y 502.754,Z 277.939,A -85,B 0,C 180,E1 -5824.989,E2 -5824.989} C_VEL
LIN {X 0,Y 505.336,Z 289.997,A -85,B 0,C 180,E1 -5826.821,E2 -5826.821} C_VEL
LIN {X 0,Y 504.641,Z 310.367,A -85,B 0,C 180,E1 -5829.629,E2 -5829.629} C_VEL
LIN {X 0,Y 503.939,Z 331.95,A -85,B 0,C 180,E1 -5832.555,E2 -5832.555} C_VEL
LIN {X 0,Y 503.623,Z 345.298,A -85,B 0,C 180,E1 -5834.34,E2 -5834.34} C_VEL
LIN {X 0,Y 505.119,Z 357.446,A -85,B 0,C 180,E1 -5834.565,E2 -5834.565} C_VEL
LIN {X 0,Y 504.544,Z 451.492,A -85,B 0,C 180,E1 -5835.946,E2 -5835.946} C_VEL
LIN {X 0,Y 504.364,Z 461.489,A -85,B 0,C 180,E1 -5836.172,E2 -5836.172} C_VEL
LIN {X 0,Y 504.148,Z 471.527,A -85,B 0,C 180,E1 -5836.5,E2 -5836.5} C_VEL
LIN {X 0,Y 503.925,Z 482.85,A -85,B 0,C 180,E1 -5837.007,E2 -5837.007} C_VEL
LIN {X 0,Y 503.651,Z 492.78,A -85,B 0,C 180,E1 -5837.574,E2 -5837.574} C_VEL
LIN {X 0,Y 503.364,Z 501.991,A -85,B 0,C 180,E1 -5838.22,E2 -5838.22} C_VEL
LIN {X 0,Y 503.071,Z 511.454,A -85,B 0,C 180,E1 -5839.03,E2 -5839.03} C_VEL
LIN {X 0,Y 502.833,Z 520.24,A -85,B 0,C 180,E1 -5839.941,E2 -5839.941} C_VEL
LIN {X 0,Y 502.625,Z 526.877,A -85,B 0,C 180,E1 -5840.749,E2 -5840.749} C_VEL
LIN {X 0,Y 502.452,Z 533.832,A -85,B 0,C 180,E1 -5841.76,E2 -5841.76} C_VEL
LIN {X 0,Y 502.3,Z 539.641,A -85,B 0,C 180,E1 -5842.768,E2 -5842.768} C_VEL
LIN {X 0,Y 502.197,Z 545.259,A -85,B 0,C 180,E1 -5843.977,E2 -5843.977} C_VEL
LIN {X 0,Y 502.111,Z 549.673,A -85,B 0,C 180,E1 -5845.185,E2 -5845.185} C_VEL
LIN {X 0,Y 502.169,Z 552.008,A -85,B 0,C 180,E1 -5845.989,E2 -5845.989} C_VEL
LIN {X 0,Y 502.117,Z 555.338,A -85,B 0,C 180,E1 -5847.595,E2 -5847.595} C_VEL
LIN {X 0,Y 501.991,Z 556.887,A -85,B 0,C 180,E1 -5849.2,E2 -5849.2} C_VEL
LIN {X 0,Y 501.989,Z 557.174,A -85,B 0,C 180,E1 -5850.002,E2 -5850.002} C_VEL
LIN {X 0,Y 502.034,Z 556.277,A -85,B 0,C 180,E1 -5851.606,E2 -5851.606} C_VEL
LIN {X 0,Y 502.117,Z 555.289,A -85,B 0,C 180,E1 -5852.408,E2 -5852.408} C_VEL
LIN {X 0,Y 502.175,Z 551.926,A -85,B 0,C 180,E1 -5854.014,E2 -5854.014} C_VEL
LIN {X 0,Y 502.179,Z 548.215,A -85,B 0,C 180,E1 -5855.22,E2 -5855.22} C_VEL
LIN {X 0,Y 502.232,Z 542.922,A -85,B 0,C 180,E1 -5856.519,E2 -5856.519} C_VEL
LIN {X 0,Y 502.35,Z 537.196,A -85,B 0,C 180,E1 -5857.638,E2 -5857.638} C_VEL
LIN {X 0,Y 502.491,Z 530.938,A -85,B 0,C 180,E1 -5858.648,E2 -5858.648} C_VEL
LIN {X 0,Y 502.678,Z 523.383,A -85,B 0,C 180,E1 -5859.659,E2 -5859.659} C_VEL
LIN {X 0,Y 502.908,Z 515.216,A -85,B 0,C 180,E1 -5860.569,E2 -5860.569} C_VEL
LIN {X 0,Y 503.187,Z 506.521,A -85,B 0,C 180,E1 -5861.379,E2 -5861.379} C_VEL
LIN {X 0,Y 503.464,Z 497.375,A -85,B 0,C 180,E1 -5862.087,E2 -5862.087} C_VEL
LIN {X 0,Y 503.747,Z 488.022,A -85,B 0,C 180,E1 -5862.685,E2 -5862.685} C_VEL
LIN {X 0,Y 504.021,Z 476.779,A -85,B 0,C 180,E1 -5863.25,E2 -5863.25} C_VEL
LIN {X 0,Y 504.249,Z 466.229,A -85,B 0,C 180,E1 -5863.655,E2 -5863.655} C_VEL
LIN {X 0,Y 504.398,Z 455.032,A -85,B 0,C 180,E1 -5863.959,E2 -5863.959} C_VEL
LIN {X 0,Y 504.639,Z 436.376,A -85,B 0,C 180,E1 -5864.261,E2 -5864.261} C_VEL
LIN {X 0,Y 504.919,Z 355.36,A -85,B 0,C 180,E1 -5865.446,E2 -5865.446} C_VEL
LIN {X 0,Y 503.55,Z 344.887,A -85,B 0,C 180,E1 -5865.65,E2 -5865.65} C_VEL
LIN {X 0,Y 504.116,Z 319.66,A -85,B 0,C 180,E1 -5868.913,E2 -5868.913} C_VEL
LIN {X 0,Y 504.601,Z 298.635,A -85,B 0,C 180,E1 -5871.659,E2 -5871.659} C_VEL
LIN {X 0,Y 504.839,Z 288.816,A -85,B 0,C 180,E1 -5872.941,E2 -5872.941} C_VEL
LIN {X 0,Y 502.783,Z 277.858,A -85,B 0,C 180,E1 -5874.477,E2 -5874.477} C_VEL
LIN {X 0,Y 502.764,Z 277.865,A -85,B 0,C 180,E1 -5877.47,E2 -5877.47} C_VEL
LIN {X 0,Y 502.793,Z 277.855,A -85,B 0,C 180,E1 -5880.211,E2 -5880.211} C_VEL
LIN {X 0,Y 502.822,Z 277.851,A -85,B 0,C 180,E1 -5883.03,E2 -5883.03} C_VEL
LIN {X 0,Y 502.763,Z 277.859,A -85,B 0,C 180,E1 -5885.95,E2 -5885.95} C_VEL
LIN {X 0,Y 502.789,Z 277.854,A -85,B 0,C 180,E1 -5888.975,E2 -5888.975} C_VEL
LIN {X 0,Y 502.815,Z 277.853,A -85,B 0,C 180,E1 -5892.134,E2 -5892.134} C_VEL
LIN {X 0,Y 502.783,Z 277.856,A -85,B 0,C 180,E1 -5895.467,E2 -5895.467} C_VEL
LIN {X 0,Y 502.807,Z 277.849,A -85,B 0,C 180,E1 -5898.933,E2 -5898.933} C_VEL
LIN {X 0,Y 502.776,Z 277.859,A -85,B 0,C 180,E1 -5902.045,E2 -5902.045} C_VEL
LIN {X 0,Y 502.788,Z 277.848,A -85,B 0,C 180,E1 -5905.034,E2 -5905.034} C_VEL
LIN {X 0,Y 502.763,Z 277.854,A -85,B 0,C 180,E1 -5907.914,E2 -5907.914} C_VEL
LIN {X 0,Y 502.812,Z 277.849,A -85,B 0,C 180,E1 -5910.712,E2 -5910.712} C_VEL
LIN {X 0,Y 502.853,Z 277.841,A -85,B 0,C 180,E1 -5913.434,E2 -5913.434} C_VEL
LIN {X 0,Y 502.795,Z 277.854,A -85,B 0,C 180,E1 -5916.087,E2 -5916.087} C_VEL
LIN {X 0,Y 502.772,Z 277.86,A -85,B 0,C 180,E1 -5918.689,E2 -5918.689} C_VEL
LIN {X 0,Y 502.813,Z 277.849,A -85,B 0,C 180,E1 -5921.877,E2 -5921.877} C_VEL
LIN {X 0,Y 502.815,Z 277.855,A -85,B 0,C 180,E1 -5924.658,E2 -5924.658} C_VEL
LIN {X 0,Y 502.866,Z 277.842,A -85,B 0,C 180,E1 -5928.026,E2 -5928.026} C_VEL
LIN {X 0,Y 502.845,Z 277.853,A -85,B 0,C 180,E1 -5931.157,E2 -5931.157} C_VEL
LIN {X 0,Y 502.871,Z 277.847,A -85,B 0,C 180,E1 -5933.581,E2 -5933.581} C_VEL
LIN {X 0,Y 502.867,Z 277.848,A -85,B 0,C 180,E1 -5936.796,E2 -5936.796} C_VEL
LIN {X 0,Y 503.151,Z 277.816,A -85,B 0,C 180,E1 -5938.9,E2 -5938.9} C_VEL
LIN {X 0,Y 503.107,Z 278.089,A -85,B 0,C 180,E1 -5939,E2 -5939} C_VEL
LIN {X 0,Y 502.965,Z 297.523,A -85,B 0,C 180,E1 -5941.602,E2 -5941.602} C_VEL
LIN {X 0,Y 502.881,Z 317.517,A -85,B 0,C 180,E1 -5944.409,E2 -5944.409} C_VEL
LIN {X 0,Y 502.859,Z 337.918,A -85,B 0,C 180,E1 -5947.428,E2 -5947.428} C_VEL
LIN {X 0,Y 504.469,Z 348.768,A -85,B 0,C 180,E1 -5947.656,E2 -5947.656} C_VEL
LIN {X 0,Y 503.946,Z 417.697,A -85,B 0,C 180,E1 -5948.741,E2 -5948.741} C_VEL
LIN {X 0,Y 503.774,Z 427.763,A -85,B 0,C 180,E1 -5949.005,E2 -5949.005} C_VEL
LIN {X 0,Y 503.636,Z 438.82,A -85,B 0,C 180,E1 -5949.438,E2 -5949.438} C_VEL
LIN {X 0,Y 503.446,Z 449.754,A -85,B 0,C 180,E1 -5950.05,E2 -5950.05} C_VEL
LIN {X 0,Y 503.156,Z 458.316,A -85,B 0,C 180,E1 -5950.666,E2 -5950.666} C_VEL
LIN {X 0,Y 502.982,Z 465.326,A -85,B 0,C 180,E1 -5951.281,E2 -5951.281} C_VEL
LIN {X 0,Y 502.8,Z 473.01,A -85,B 0,C 180,E1 -5952.103,E2 -5952.103} C_VEL
LIN {X 0,Y 502.6,Z 479.349,A -85,B 0,C 180,E1 -5952.929,E2 -5952.929} C_VEL
LIN {X 0,Y 502.457,Z 484.598,A -85,B 0,C 180,E1 -5953.756,E2 -5953.756} C_VEL
LIN {X 0,Y 502.347,Z 488.953,A -85,B 0,C 180,E1 -5954.586,E2 -5954.586} C_VEL
LIN {X 0,Y 502.276,Z 492.546,A -85,B 0,C 180,E1 -5955.418,E2 -5955.418} C_VEL
LIN {X 0,Y 502.185,Z 496.668,A -85,B 0,C 180,E1 -5956.673,E2 -5956.673} C_VEL
LIN {X 0,Y 502.092,Z 499.465,A -85,B 0,C 180,E1 -5957.936,E2 -5957.936} C_VEL
LIN {X 0,Y 502.038,Z 500.524,A -85,B 0,C 180,E1 -5958.783,E2 -5958.783} C_VEL
LIN {X 0,Y 502.038,Z 501.035,A -85,B 0,C 180,E1 -5959.632,E2 -5959.632} C_VEL
LIN {X 0,Y 502.046,Z 501.008,A -85,B 0,C 180,E1 -5960.486,E2 -5960.486} C_VEL
LIN {X 0,Y 502.082,Z 500.434,A -85,B 0,C 180,E1 -5961.343,E2 -5961.343} C_VEL
LIN {X 0,Y 502.094,Z 498.658,A -85,B 0,C 180,E1 -5962.518,E2 -5962.518} C_VEL
LIN {X 0,Y 502.202,Z 496.296,A -85,B 0,C 180,E1 -5963.506,E2 -5963.506} C_VEL
LIN {X 0,Y 502.245,Z 492.802,A -85,B 0,C 180,E1 -5964.565,E2 -5964.565} C_VEL
LIN {X 0,Y 502.365,Z 487.823,A -85,B 0,C 180,E1 -5965.702,E2 -5965.702} C_VEL
LIN {X 0,Y 502.54,Z 481.567,A -85,B 0,C 180,E1 -5966.809,E2 -5966.809} C_VEL
LIN {X 0,Y 502.677,Z 475.166,A -85,B 0,C 180,E1 -5967.703,E2 -5967.703} C_VEL
LIN {X 0,Y 502.878,Z 467.173,A -85,B 0,C 180,E1 -5968.599,E2 -5968.599} C_VEL
LIN {X 0,Y 503.116,Z 459.873,A -85,B 0,C 180,E1 -5969.27,E2 -5969.27} C_VEL
LIN {X 0,Y 503.318,Z 452.504,A -85,B 0,C 180,E1 -5969.832,E2 -5969.832} C_VEL
LIN {X 0,Y 503.47,Z 444.322,A -85,B 0,C 180,E1 -5970.342,E2 -5970.342} C_VEL
LIN {X 0,Y 503.676,Z 435.058,A -85,B 0,C 180,E1 -5970.792,E2 -5970.792} C_VEL
LIN {X 0,Y 503.811,Z 425.832,A -85,B 0,C 180,E1 -5971.126,E2 -5971.126} C_VEL
LIN {X 0,Y 503.877,Z 416.609,A -85,B 0,C 180,E1 -5971.355,E2 -5971.355} C_VEL
LIN {X 0,Y 504.339,Z 348.565,A -85,B 0,C 180,E1 -5972.398,E2 -5972.398} C_VEL
LIN {X 0,Y 503.554,Z 343.313,A -85,B 0,C 180,E1 -5972.501,E2 -5972.501} C_VEL
LIN {X 0,Y 502.767,Z 340.169,A -85,B 0,C 180,E1 -5972.648,E2 -5972.648} C_VEL
LIN {X 0,Y 501.644,Z 337.651,A -85,B 0,C 180,E1 -5972.905,E2 -5972.905} C_VEL
LIN {X 0,Y 499.192,Z 333.803,A -85,B 0,C 180,E1 -5973.583,E2 -5973.583} C_VEL
LIN {X 0,Y 496.977,Z 329.492,A -85,B 0,C 180,E1 -5974.434,E2 -5974.434} C_VEL
LIN {X 0,Y 496.167,Z 326.022,A -85,B 0,C 180,E1 -5975.078,E2 -5975.078} C_VEL
LIN {X 0,Y 496.128,Z 324.832,A -85,B 0,C 180,E1 -5975.292,E2 -5975.292} C_VEL
LIN {X 0,Y 496.603,Z 308.423,A -85,B 0,C 180,E1 -5978.255,E2 -5978.255} C_VEL
LIN {X 0,Y 496.995,Z 290.915,A -85,B 0,C 180,E1 -5981.459,E2 -5981.459} C_VEL
LIN {X 0,Y 497.034,Z 285.692,A -85,B 0,C 180,E1 -5982.427,E2 -5982.427} C_VEL
LIN {X 0,Y 495.747,Z 278.734,A -85,B 0,C 180,E1 -5983.817,E2 -5983.817} C_VEL
LIN {X 0,Y 495.714,Z 278.739,A -85,B 0,C 180,E1 -5987.119,E2 -5987.119} C_VEL
LIN {X 0,Y 495.745,Z 278.729,A -85,B 0,C 180,E1 -5989.956,E2 -5989.956} C_VEL
LIN {X 0,Y 495.699,Z 278.732,A -85,B 0,C 180,E1 -5992.558,E2 -5992.558} C_VEL
LIN {X 0,Y 495.763,Z 278.729,A -85,B 0,C 180,E1 -5995.458,E2 -5995.458} C_VEL
LIN {X 0,Y 495.75,Z 278.729,A -85,B 0,C 180,E1 -5998.365,E2 -5998.365} C_VEL
LIN {X 0,Y 495.724,Z 278.729,A -85,B 0,C 180,E1 -6001.183,E2 -6001.183} C_VEL
LIN {X 0,Y 495.717,Z 278.735,A -85,B 0,C 180,E1 -6003.929,E2 -6003.929} C_VEL
LIN {X 0,Y 495.745,Z 278.727,A -85,B 0,C 180,E1 -6007.145,E2 -6007.145} C_VEL
LIN {X 0,Y 495.757,Z 278.728,A -85,B 0,C 180,E1 -6010.109,E2 -6010.109} C_VEL
LIN {X 0,Y 495.754,Z 278.735,A -85,B 0,C 180,E1 -6012.68,E2 -6012.68} C_VEL
LIN {X 0,Y 495.779,Z 278.727,A -85,B 0,C 180,E1 -6015.217,E2 -6015.217} C_VEL
LIN {X 0,Y 495.853,Z 278.715,A -85,B 0,C 180,E1 -6018.554,E2 -6018.554} C_VEL
LIN {X 0,Y 495.815,Z 278.72,A -85,B 0,C 180,E1 -6021.85,E2 -6021.85} C_VEL
LIN {X 0,Y 495.856,Z 278.713,A -85,B 0,C 180,E1 -6024.305,E2 -6024.305} C_VEL
LIN {X 0,Y 495.977,Z 278.707,A -85,B 0,C 180,E1 -6027.562,E2 -6027.562} C_VEL
LIN {X 0,Y 495.975,Z 278.703,A -85,B 0,C 180,E1 -6029.998,E2 -6029.998} C_VEL
LIN {X 0,Y 495.977,Z 278.7,A -85,B 0,C 180,E1 -6032.434,E2 -6032.434} C_VEL
LIN {X 0,Y 495.853,Z 278.717,A -85,B 0,C 180,E1 -6035.692,E2 -6035.692} C_VEL
LIN {X 0,Y 495.811,Z 278.728,A -85,B 0,C 180,E1 -6038.147,E2 -6038.147} C_VEL
LIN {X 0,Y 495.847,Z 278.714,A -85,B 0,C 180,E1 -6041.442,E2 -6041.442} C_VEL
LIN {X 0,Y 495.775,Z 278.729,A -85,B 0,C 180,E1 -6044.78,E2 -6044.78} C_VEL
LIN {X 0,Y 495.752,Z 278.727,A -85,B 0,C 180,E1 -6047.316,E2 -6047.316} C_VEL
LIN {X 0,Y 495.753,Z 278.725,A -85,B 0,C 180,E1 -6049.887,E2 -6049.887} C_VEL
LIN {X 0,Y 495.748,Z 278.733,A -85,B 0,C 180,E1 -6052.856,E2 -6052.856} C_VEL
LIN {X 0,Y 495.711,Z 278.731,A -85,B 0,C 180,E1 -6056.068,E2 -6056.068} C_VEL
LIN {X 0,Y 495.728,Z 278.73,A -85,B 0,C 180,E1 -6058.813,E2 -6058.813} C_VEL
LIN {X 0,Y 495.736,Z 278.735,A -85,B 0,C 180,E1 -6061.721,E2 -6061.721} C_VEL
LIN {X 0,Y 495.748,Z 278.726,A -85,B 0,C 180,E1 -6064.69,E2 -6064.69} C_VEL
LIN {X 0,Y 495.705,Z 278.736,A -85,B 0,C 180,E1 -6067.557,E2 -6067.557} C_VEL
LIN {X 0,Y 495.739,Z 278.729,A -85,B 0,C 180,E1 -6070.696,E2 -6070.696} C_VEL
LIN {X 0,Y 495.696,Z 278.738,A -85,B 0,C 180,E1 -6073.997,E2 -6073.997} C_VEL
LIN {X 0,Y 495.691,Z 278.734,A -85,B 0,C 180,E1 -6077.113,E2 -6077.113} C_VEL
LIN {X 0,Y 495.721,Z 278.731,A -85,B 0,C 180,E1 -6079.949,E2 -6079.949} C_VEL
LIN {X 0,Y 495.689,Z 278.74,A -85,B 0,C 180,E1 -6082.549,E2 -6082.549} C_VEL
LIN {X 0,Y 495.733,Z 278.73,A -85,B 0,C 180,E1 -6085.453,E2 -6085.453} C_VEL
LIN {X 0,Y 495.708,Z 278.732,A -85,B 0,C 180,E1 -6088.36,E2 -6088.36} C_VEL
LIN {X 0,Y 495.743,Z 278.733,A -85,B 0,C 180,E1 -6091.503,E2 -6091.503} C_VEL
LIN {X 0,Y 495.748,Z 278.728,A -85,B 0,C 180,E1 -6093.929,E2 -6093.929} C_VEL
LIN {X 0,Y 495.712,Z 278.734,A -85,B 0,C 180,E1 -6097.135,E2 -6097.135} C_VEL
LIN {X 0,Y 495.716,Z 278.734,A -85,B 0,C 180,E1 -6100.107,E2 -6100.107} C_VEL
LIN {X 0,Y 495.73,Z 278.729,A -85,B 0,C 180,E1 -6102.679,E2 -6102.679} C_VEL
LIN {X 0,Y 495.737,Z 278.728,A -85,B 0,C 180,E1 -6105.215,E2 -6105.215} C_VEL
LIN {X 0,Y 495.813,Z 278.723,A -85,B 0,C 180,E1 -6108.553,E2 -6108.553} C_VEL
LIN {X 0,Y 495.813,Z 278.72,A -85,B 0,C 180,E1 -6111.851,E2 -6111.851} C_VEL
LIN {X 0,Y 495.857,Z 278.718,A -85,B 0,C 180,E1 -6114.306,E2 -6114.306} C_VEL
LIN {X 0,Y 495.935,Z 278.703,A -85,B 0,C 180,E1 -6117.563,E2 -6117.563} C_VEL
LIN {X 0,Y 495.93,Z 278.703,A -85,B 0,C 180,E1 -6120,E2 -6120} C_VEL
LIN {X 0,Y 495.934,Z 278.705,A -85,B 0,C 180,E1 -6122.436,E2 -6122.436} C_VEL
LIN {X 0,Y 495.856,Z 278.716,A -85,B 0,C 180,E1 -6125.693,E2 -6125.693} C_VEL
LIN {X 0,Y 495.812,Z 278.719,A -85,B 0,C 180,E1 -6128.149,E2 -6128.149} C_VEL
LIN {X 0,Y 495.811,Z 278.727,A -85,B 0,C 180,E1 -6131.446,E2 -6131.446} C_VEL
LIN {X 0,Y 495.735,Z 278.728,A -85,B 0,C 180,E1 -6134.784,E2 -6134.784} C_VEL
LIN {X 0,Y 495.737,Z 278.733,A -85,B 0,C 180,E1 -6138.173,E2 -6138.173} C_VEL
LIN {X 0,Y 495.719,Z 278.731,A -85,B 0,C 180,E1 -6140.758,E2 -6140.758} C_VEL
LIN {X 0,Y 495.709,Z 278.731,A -85,B 0,C 180,E1 -6143.389,E2 -6143.389} C_VEL
LIN {X 0,Y 495.737,Z 278.732,A -85,B 0,C 180,E1 -6146.07,E2 -6146.07} C_VEL
LIN {X 0,Y 495.72,Z 278.735,A -85,B 0,C 180,E1 -6148.818,E2 -6148.818} C_VEL
LIN {X 0,Y 495.703,Z 278.732,A -85,B 0,C 180,E1 -6151.728,E2 -6151.728} C_VEL
LIN {X 0,Y 495.727,Z 278.736,A -85,B 0,C 180,E1 -6154.698,E2 -6154.698} C_VEL
LIN {X 0,Y 495.684,Z 278.736,A -85,B 0,C 180,E1 -6157.565,E2 -6157.565} C_VEL
LIN {X 0,Y 495.711,Z 278.733,A -85,B 0,C 180,E1 -6160.705,E2 -6160.705} C_VEL
LIN {X 0,Y 495.679,Z 278.74,A -85,B 0,C 180,E1 -6163.697,E2 -6163.697} C_VEL
LIN {X 0,Y 495.689,Z 278.734,A -85,B 0,C 180,E1 -6166.31,E2 -6166.31} C_VEL
LIN {X 0,Y 495.732,Z 278.732,A -85,B 0,C 180,E1 -6169.304,E2 -6169.304} C_VEL
LIN {X 0,Y 495.676,Z 278.737,A -85,B 0,C 180,E1 -6172.44,E2 -6172.44} C_VEL
LIN {X 0,Y 495.738,Z 278.729,A -85,B 0,C 180,E1 -6175.46,E2 -6175.46} C_VEL
LIN {X 0,Y 495.723,Z 278.737,A -85,B 0,C 180,E1 -6178.367,E2 -6178.367} C_VEL
LIN {X 0,Y 495.702,Z 278.735,A -85,B 0,C 180,E1 -6181.186,E2 -6181.186} C_VEL
LIN {X 0,Y 495.718,Z 278.739,A -85,B 0,C 180,E1 -6184.384,E2 -6184.384} C_VEL
LIN {X 0,Y 495.748,Z 278.909,A -85,B 0,C 180,E1 -6184.779,E2 -6184.779} C_VEL
LIN {X 0,Y 498.45,Z 291.703,A -85,B 0,C 180,E1 -6186.751,E2 -6186.751} C_VEL
LIN {X 0,Y 497.689,Z 311.72,A -85,B 0,C 180,E1 -6189.547,E2 -6189.547} C_VEL
LIN {X 0,Y 496.957,Z 333.295,A -85,B 0,C 180,E1 -6192.515,E2 -6192.515} C_VEL
LIN {X 0,Y 496.629,Z 345.284,A -85,B 0,C 180,E1 -6194.136,E2 -6194.136} C_VEL
LIN {X 0,Y 498.232,Z 358.29,A -85,B 0,C 180,E1 -6194.38,E2 -6194.38} C_VEL
LIN {X 0,Y 497.63,Z 451.309,A -85,B 0,C 180,E1 -6195.772,E2 -6195.772} C_VEL
LIN {X 0,Y 497.434,Z 461.276,A -85,B 0,C 180,E1 -6196.001,E2 -6196.001} C_VEL
LIN {X 0,Y 497.189,Z 471.906,A -85,B 0,C 180,E1 -6196.359,E2 -6196.359} C_VEL
LIN {X 0,Y 496.94,Z 482.133,A -85,B 0,C 180,E1 -6196.821,E2 -6196.821} C_VEL
LIN {X 0,Y 496.641,Z 492.739,A -85,B 0,C 180,E1 -6197.437,E2 -6197.437} C_VEL
LIN {X 0,Y 496.321,Z 502.658,A -85,B 0,C 180,E1 -6198.154,E2 -6198.154} C_VEL
LIN {X 0,Y 496.073,Z 510.925,A -85,B 0,C 180,E1 -6198.873,E2 -6198.873} C_VEL
LIN {X 0,Y 495.799,Z 519.743,A -85,B 0,C 180,E1 -6199.797,E2 -6199.797} C_VEL
LIN {X 0,Y 495.577,Z 526.406,A -85,B 0,C 180,E1 -6200.617,E2 -6200.617} C_VEL
LIN {X 0,Y 495.372,Z 533.381,A -85,B 0,C 180,E1 -6201.641,E2 -6201.641} C_VEL
LIN {X 0,Y 495.241,Z 539.209,A -85,B 0,C 180,E1 -6202.665,E2 -6202.665} C_VEL
LIN {X 0,Y 495.099,Z 545.376,A -85,B 0,C 180,E1 -6204.033,E2 -6204.033} C_VEL
LIN {X 0,Y 495.038,Z 549.266,A -85,B 0,C 180,E1 -6205.116,E2 -6205.116} C_VEL
LIN {X 0,Y 495.062,Z 551.601,A -85,B 0,C 180,E1 -6205.932,E2 -6205.932} C_VEL
LIN {X 0,Y 495.05,Z 554.945,A -85,B 0,C 180,E1 -6207.561,E2 -6207.561} C_VEL
LIN {X 0,Y 494.911,Z 556.493,A -85,B 0,C 180,E1 -6209.188,E2 -6209.188} C_VEL
LIN {X 0,Y 494.906,Z 556.78,A -85,B 0,C 180,E1 -6210.002,E2 -6210.002} C_VEL
LIN {X 0,Y 494.96,Z 555.877,A -85,B 0,C 180,E1 -6211.629,E2 -6211.629} C_VEL
LIN {X 0,Y 495.05,Z 554.885,A -85,B 0,C 180,E1 -6212.442,E2 -6212.442} C_VEL
LIN {X 0,Y 495.07,Z 551.502,A -85,B 0,C 180,E1 -6214.072,E2 -6214.072} C_VEL
LIN {X 0,Y 495.11,Z 547.776,A -85,B 0,C 180,E1 -6215.295,E2 -6215.295} C_VEL
LIN {X 0,Y 495.16,Z 542.897,A -85,B 0,C 180,E1 -6216.521,E2 -6216.521} C_VEL
LIN {X 0,Y 495.262,Z 536.706,A -85,B 0,C 180,E1 -6217.748,E2 -6217.748} C_VEL
LIN {X 0,Y 495.427,Z 530.421,A -85,B 0,C 180,E1 -6218.772,E2 -6218.772} C_VEL
LIN {X 0,Y 495.624,Z 522.829,A -85,B 0,C 180,E1 -6219.798,E2 -6219.798} C_VEL
LIN {X 0,Y 495.826,Z 514.616,A -85,B 0,C 180,E1 -6220.722,E2 -6220.722} C_VEL
LIN {X 0,Y 496.141,Z 507.128,A -85,B 0,C 180,E1 -6221.439,E2 -6221.439} C_VEL
LIN {X 0,Y 496.442,Z 496.674,A -85,B 0,C 180,E1 -6222.261,E2 -6222.261} C_VEL
LIN {X 0,Y 496.771,Z 487.072,A -85,B 0,C 180,E1 -6222.875,E2 -6222.875} C_VEL
LIN {X 0,Y 497.041,Z 477.097,A -85,B 0,C 180,E1 -6223.388,E2 -6223.388} C_VEL
LIN {X 0,Y 497.321,Z 465.96,A -85,B 0,C 180,E1 -6223.823,E2 -6223.823} C_VEL
LIN {X 0,Y 497.46,Z 454.792,A -85,B 0,C 180,E1 -6224.132,E2 -6224.132} C_VEL
LIN {X 0,Y 497.723,Z 436.185,A -85,B 0,C 180,E1 -6224.437,E2 -6224.437} C_VEL
LIN {X 0,Y 498.059,Z 356.351,A -85,B 0,C 180,E1 -6225.626,E2 -6225.626} C_VEL
LIN {X 0,Y 496.555,Z 344.733,A -85,B 0,C 180,E1 -6225.863,E2 -6225.863} C_VEL
LIN {X 0,Y 497.168,Z 319.404,A -85,B 0,C 180,E1 -6229.187,E2 -6229.187} C_VEL
LIN {X 0,Y 497.692,Z 299.93,A -85,B 0,C 180,E1 -6231.757,E2 -6231.757} C_VEL
LIN {X 0,Y 497.927,Z 290.077,A -85,B 0,C 180,E1 -6233.058,E2 -6233.058} C_VEL
LIN {X 0,Y 495.733,Z 278.736,A -85,B 0,C 180,E1 -6234.698,E2 -6234.698} C_VEL
LIN {X 0,Y 495.706,Z 278.742,A -85,B 0,C 180,E1 -6237.895,E2 -6237.895} C_VEL
LIN {X 0,Y 495.738,Z 278.734,A -85,B 0,C 180,E1 -6240.687,E2 -6240.687} C_VEL
LIN {X 0,Y 495.749,Z 278.736,A -85,B 0,C 180,E1 -6243.563,E2 -6243.563} C_VEL
LIN {X 0,Y 495.717,Z 278.733,A -85,B 0,C 180,E1 -6246.543,E2 -6246.543} C_VEL
LIN {X 0,Y 495.743,Z 278.738,A -85,B 0,C 180,E1 -6249.637,E2 -6249.637} C_VEL
LIN {X 0,Y 495.725,Z 278.733,A -85,B 0,C 180,E1 -6252.506,E2 -6252.506} C_VEL
LIN {X 0,Y 495.732,Z 278.732,A -85,B 0,C 180,E1 -6255.138,E2 -6255.138} C_VEL
LIN {X 0,Y 495.741,Z 278.735,A -85,B 0,C 180,E1 -6258.218,E2 -6258.218} C_VEL
LIN {X 0,Y 495.748,Z 278.728,A -85,B 0,C 180,E1 -6261.229,E2 -6261.229} C_VEL
LIN {X 0,Y 495.738,Z 278.731,A -85,B 0,C 180,E1 -6264.462,E2 -6264.462} C_VEL
LIN {X 0,Y 495.745,Z 278.724,A -85,B 0,C 180,E1 -6267.404,E2 -6267.404} C_VEL
LIN {X 0,Y 495.755,Z 278.731,A -85,B 0,C 180,E1 -6270.253,E2 -6270.253} C_VEL
LIN {X 0,Y 495.806,Z 278.72,A -85,B 0,C 180,E1 -6273.247,E2 -6273.247} C_VEL
LIN {X 0,Y 495.748,Z 278.729,A -85,B 0,C 180,E1 -6275.725,E2 -6275.725} C_VEL
LIN {X 0,Y 495.737,Z 278.736,A -85,B 0,C 180,E1 -6278.371,E2 -6278.371} C_VEL
LIN {X 0,Y 495.753,Z 278.733,A -85,B 0,C 180,E1 -6280.971,E2 -6280.971} C_VEL
LIN {X 0,Y 495.752,Z 278.729,A -85,B 0,C 180,E1 -6283.53,E2 -6283.53} C_VEL
LIN {X 0,Y 495.775,Z 278.726,A -85,B 0,C 180,E1 -6286.056,E2 -6286.056} C_VEL
LIN {X 0,Y 495.841,Z 278.722,A -85,B 0,C 180,E1 -6288.555,E2 -6288.555} C_VEL
LIN {X 0,Y 495.84,Z 278.721,A -85,B 0,C 180,E1 -6291.852,E2 -6291.852} C_VEL
LIN {X 0,Y 495.863,Z 278.719,A -85,B 0,C 180,E1 -6294.307,E2 -6294.307} C_VEL
LIN {X 0,Y 496.16,Z 278.686,A -85,B 0,C 180,E1 -6298.783,E2 -6298.783} C_VEL
LIN {X 0,Y 496.114,Z 278.783,A -85,B 0,C 180,E1 -6298.884,E2 -6298.884} C_VEL
LIN {X 0,Y 495.942,Z 300.587,A -85,B 0,C 180,E1 -6301.828,E2 -6301.828} C_VEL
LIN {X 0,Y 495.874,Z 320.714,A -85,B 0,C 180,E1 -6304.675,E2 -6304.675} C_VEL
LIN {X 0,Y 495.863,Z 337.964,A -85,B 0,C 180,E1 -6307.226,E2 -6307.226} C_VEL
LIN {X 0,Y 497.598,Z 350.112,A -85,B 0,C 180,E1 -6307.475,E2 -6307.475} C_VEL
LIN {X 0,Y 497.035,Z 418.807,A -85,B 0,C 180,E1 -6308.589,E2 -6308.589} C_VEL
LIN {X 0,Y 496.879,Z 429.086,A -85,B 0,C 180,E1 -6308.874,E2 -6308.874} C_VEL
LIN {X 0,Y 496.664,Z 440.835,A -85,B 0,C 180,E1 -6309.366,E2 -6309.366} C_VEL
LIN {X 0,Y 496.431,Z 451.322,A -85,B 0,C 180,E1 -6309.987,E2 -6309.987} C_VEL
LIN {X 0,Y 496.144,Z 459.657,A -85,B 0,C 180,E1 -6310.612,E2 -6310.612} C_VEL
LIN {X 0,Y 495.939,Z 467.537,A -85,B 0,C 180,E1 -6311.34,E2 -6311.34} C_VEL
LIN {X 0,Y 495.717,Z 475.797,A -85,B 0,C 180,E1 -6312.279,E2 -6312.279} C_VEL
LIN {X 0,Y 495.492,Z 483.022,A -85,B 0,C 180,E1 -6313.326,E2 -6313.326} C_VEL
LIN {X 0,Y 495.325,Z 488.727,A -85,B 0,C 180,E1 -6314.377,E2 -6314.377} C_VEL
LIN {X 0,Y 495.21,Z 494.02,A -85,B 0,C 180,E1 -6315.644,E2 -6315.644} C_VEL
LIN {X 0,Y 495.091,Z 497.879,A -85,B 0,C 180,E1 -6316.919,E2 -6316.919} C_VEL
LIN {X 0,Y 494.995,Z 500.265,A -85,B 0,C 180,E1 -6318.202,E2 -6318.202} C_VEL
LIN {X 0,Y 494.954,Z 501.215,A -85,B 0,C 180,E1 -6319.062,E2 -6319.062} C_VEL
LIN {X 0,Y 494.977,Z 501.424,A -85,B 0,C 180,E1 -6320.439,E2 -6320.439} C_VEL
LIN {X 0,Y 494.986,Z 500.457,A -85,B 0,C 180,E1 -6321.664,E2 -6321.664} C_VEL
LIN {X 0,Y 495.03,Z 498.804,A -85,B 0,C 180,E1 -6322.669,E2 -6322.669} C_VEL
LIN {X 0,Y 495.141,Z 495.788,A -85,B 0,C 180,E1 -6323.862,E2 -6323.862} C_VEL
LIN {X 0,Y 495.241,Z 490.939,A -85,B 0,C 180,E1 -6325.198,E2 -6325.198} C_VEL
LIN {X 0,Y 495.42,Z 484.961,A -85,B 0,C 180,E1 -6326.383,E2 -6326.383} C_VEL
LIN {X 0,Y 495.533,Z 479.747,A -85,B 0,C 180,E1 -6327.219,E2 -6327.219} C_VEL
LIN {X 0,Y 495.731,Z 473.193,A -85,B 0,C 180,E1 -6328.085,E2 -6328.085} C_VEL
LIN {X 0,Y 495.88,Z 466.599,A -85,B 0,C 180,E1 -6328.808,E2 -6328.808} C_VEL
LIN {X 0,Y 496.14,Z 459.108,A -85,B 0,C 180,E1 -6329.489,E2 -6329.489} C_VEL
LIN {X 0,Y 496.361,Z 451.327,A -85,B 0,C 180,E1 -6330.071,E2 -6330.071} C_VEL
LIN {X 0,Y 496.527,Z 443.967,A -85,B 0,C 180,E1 -6330.523,E2 -6330.523} C_VEL
LIN {X 0,Y 496.72,Z 434.635,A -85,B 0,C 180,E1 -6330.975,E2 -6330.975} C_VEL
LIN {X 0,Y 496.876,Z 424.984,A -85,B 0,C 180,E1 -6331.32,E2 -6331.32} C_VEL
LIN {X 0,Y 497.015,Z 413.485,A -85,B 0,C 180,E1 -6331.585,E2 -6331.585} C_VEL
LIN {X 0,Y 497.362,Z 348.611,A -85,B 0,C 180,E1 -6332.587,E2 -6332.587} C_VEL
LIN {X 0,Y 495.868,Z 338.818,A -85,B 0,C 180,E1 -6332.793,E2 -6332.793} C_VEL
LIN {X 0,Y 496.128,Z 324.832,A -85,B 0,C 180,E1 -6335.292,E2 -6335.292} C_VEL
LIN {X 0,Y 495.563,Z 321.741,A -85,B 0,C 180,E1 -6335.87,E2 -6335.87} C_VEL
LIN {X 0,Y 490.233,Z 312.219,A -85,B 0,C 180,E1 -6337.8,E2 -6337.8} C_VEL
LIN {X 0,Y 489.63,Z 309.134,A -85,B 0,C 180,E1 -6338.389,E2 -6338.389} C_VEL
LIN {X 0,Y 490.104,Z 290.786,A -85,B 0,C 180,E1 -6341.787,E2 -6341.787} C_VEL
LIN {X 0,Y 489.965,Z 286.134,A -85,B 0,C 180,E1 -6342.671,E2 -6342.671} C_VEL
LIN {X 0,Y 488.701,Z 279.611,A -85,B 0,C 180,E1 -6343.988,E2 -6343.988} C_VEL
LIN {X 0,Y 488.674,Z 279.616,A -85,B 0,C 180,E1 -6347.179,E2 -6347.179} C_VEL
LIN {X 0,Y 488.725,Z 279.608,A -85,B 0,C 180,E1 -6349.678,E2 -6349.678} C_VEL
LIN {X 0,Y 488.653,Z 279.61,A -85,B 0,C 180,E1 -6352.841,E2 -6352.841} C_VEL
LIN {X 0,Y 488.714,Z 279.611,A -85,B 0,C 180,E1 -6355.888,E2 -6355.888} C_VEL
LIN {X 0,Y 488.685,Z 279.606,A -85,B 0,C 180,E1 -6358.821,E2 -6358.821} C_VEL
LIN {X 0,Y 488.692,Z 279.608,A -85,B 0,C 180,E1 -6361.669,E2 -6361.669} C_VEL
LIN {X 0,Y 488.698,Z 279.605,A -85,B 0,C 180,E1 -6364.96,E2 -6364.96} C_VEL
LIN {X 0,Y 488.688,Z 279.609,A -85,B 0,C 180,E1 -6368.043,E2 -6368.043} C_VEL
LIN {X 0,Y 488.733,Z 279.609,A -85,B 0,C 180,E1 -6370.687,E2 -6370.687} C_VEL
LIN {X 0,Y 488.759,Z 279.598,A -85,B 0,C 180,E1 -6374.145,E2 -6374.145} C_VEL
LIN {X 0,Y 488.74,Z 279.601,A -85,B 0,C 180,E1 -6377.543,E2 -6377.543} C_VEL
LIN {X 0,Y 488.744,Z 279.599,A -85,B 0,C 180,E1 -6380.063,E2 -6380.063} C_VEL
LIN {X 0,Y 488.824,Z 279.591,A -85,B 0,C 180,E1 -6382.768,E2 -6382.768} C_VEL
LIN {X 0,Y 488.792,Z 279.596,A -85,B 0,C 180,E1 -6385.05,E2 -6385.05} C_VEL
LIN {X 0,Y 488.943,Z 279.583,A -85,B 0,C 180,E1 -6387.527,E2 -6387.527} C_VEL
LIN {X 0,Y 488.944,Z 279.579,A -85,B 0,C 180,E1 -6389.998,E2 -6389.998} C_VEL
LIN {X 0,Y 488.943,Z 279.576,A -85,B 0,C 180,E1 -6392.47,E2 -6392.47} C_VEL
LIN {X 0,Y 488.812,Z 279.595,A -85,B 0,C 180,E1 -6395.774,E2 -6395.774} C_VEL
LIN {X 0,Y 488.757,Z 279.606,A -85,B 0,C 180,E1 -6398.265,E2 -6398.265} C_VEL
LIN {X 0,Y 488.803,Z 279.592,A -85,B 0,C 180,E1 -6401.61,E2 -6401.61} C_VEL
LIN {X 0,Y 488.752,Z 279.601,A -85,B 0,C 180,E1 -6404.997,E2 -6404.997} C_VEL
LIN {X 0,Y 488.739,Z 279.604,A -85,B 0,C 180,E1 -6408.439,E2 -6408.439} C_VEL
LIN {X 0,Y 488.699,Z 279.612,A -85,B 0,C 180,E1 -6411.067,E2 -6411.067} C_VEL
LIN {X 0,Y 488.658,Z 279.611,A -85,B 0,C 180,E1 -6413.743,E2 -6413.743} C_VEL
LIN {X 0,Y 488.689,Z 279.61,A -85,B 0,C 180,E1 -6416.918,E2 -6416.918} C_VEL
LIN {X 0,Y 488.706,Z 279.604,A -85,B 0,C 180,E1 -6420.215,E2 -6420.215} C_VEL
LIN {X 0,Y 488.715,Z 279.609,A -85,B 0,C 180,E1 -6423.48,E2 -6423.48} C_VEL
LIN {X 0,Y 488.66,Z 279.611,A -85,B 0,C 180,E1 -6426.35,E2 -6426.35} C_VEL
LIN {X 0,Y 488.674,Z 279.608,A -85,B 0,C 180,E1 -6429.25,E2 -6429.25} C_VEL
LIN {X 0,Y 488.679,Z 279.609,A -85,B 0,C 180,E1 -6431.595,E2 -6431.595} C_VEL
LIN {X 0,Y 488.669,Z 279.611,A -85,B 0,C 180,E1 -6434.798,E2 -6434.798} C_VEL
LIN {X 0,Y 488.657,Z 279.609,A -85,B 0,C 180,E1 -6437.47,E2 -6437.47} C_VEL
LIN {X 0,Y 488.697,Z 279.605,A -85,B 0,C 180,E1 -6439.672,E2 -6439.672} C_VEL
LIN {X 0,Y 488.64,Z 279.62,A -85,B 0,C 180,E1 -6442.837,E2 -6442.837} C_VEL
LIN {X 0,Y 488.68,Z 279.607,A -85,B 0,C 180,E1 -6445.883,E2 -6445.883} C_VEL
LIN {X 0,Y 488.647,Z 279.616,A -85,B 0,C 180,E1 -6448.817,E2 -6448.817} C_VEL
LIN {X 0,Y 488.699,Z 279.608,A -85,B 0,C 180,E1 -6451.668,E2 -6451.668} C_VEL
LIN {X 0,Y 488.7,Z 279.604,A -85,B 0,C 180,E1 -6454.441,E2 -6454.441} C_VEL
LIN {X 0,Y 488.674,Z 279.611,A -85,B 0,C 180,E1 -6457.15,E2 -6457.15} C_VEL
LIN {X 0,Y 488.67,Z 279.617,A -85,B 0,C 180,E1 -6459.808,E2 -6459.808} C_VEL
LIN {X 0,Y 488.677,Z 279.609,A -85,B 0,C 180,E1 -6462.421,E2 -6462.421} C_VEL
LIN {X 0,Y 488.707,Z 279.603,A -85,B 0,C 180,E1 -6464.997,E2 -6464.997} C_VEL
LIN {X 0,Y 488.772,Z 279.602,A -85,B 0,C 180,E1 -6468.386,E2 -6468.386} C_VEL
LIN {X 0,Y 488.757,Z 279.598,A -85,B 0,C 180,E1 -6471.732,E2 -6471.732} C_VEL
LIN {X 0,Y 488.813,Z 279.595,A -85,B 0,C 180,E1 -6474.223,E2 -6474.223} C_VEL
LIN {X 0,Y 488.904,Z 279.579,A -85,B 0,C 180,E1 -6477.528,E2 -6477.528} C_VEL
LIN {X 0,Y 488.902,Z 279.579,A -85,B 0,C 180,E1 -6480,E2 -6480} C_VEL
LIN {X 0,Y 488.903,Z 279.581,A -85,B 0,C 180,E1 -6482.471,E2 -6482.471} C_VEL
LIN {X 0,Y 488.812,Z 279.592,A -85,B 0,C 180,E1 -6485.776,E2 -6485.776} C_VEL
LIN {X 0,Y 488.756,Z 279.597,A -85,B 0,C 180,E1 -6488.267,E2 -6488.267} C_VEL
LIN {X 0,Y 488.77,Z 279.605,A -85,B 0,C 180,E1 -6491.613,E2 -6491.613} C_VEL
LIN {X 0,Y 488.705,Z 279.604,A -85,B 0,C 180,E1 -6495.002,E2 -6495.002} C_VEL
LIN {X 0,Y 488.697,Z 279.607,A -85,B 0,C 180,E1 -6498.444,E2 -6498.444} C_VEL
LIN {X 0,Y 488.657,Z 279.609,A -85,B 0,C 180,E1 -6501.073,E2 -6501.073} C_VEL
LIN {X 0,Y 488.648,Z 279.613,A -85,B 0,C 180,E1 -6503.747,E2 -6503.747} C_VEL
LIN {X 0,Y 488.739,Z 279.602,A -85,B 0,C 180,E1 -6506.946,E2 -6506.946} C_VEL
LIN {X 0,Y 488.658,Z 279.615,A -85,B 0,C 180,E1 -6510.365,E2 -6510.365} C_VEL
LIN {X 0,Y 488.687,Z 279.607,A -85,B 0,C 180,E1 -6513.487,E2 -6513.487} C_VEL
LIN {X 0,Y 488.641,Z 279.613,A -85,B 0,C 180,E1 -6516.359,E2 -6516.359} C_VEL
LIN {X 0,Y 488.657,Z 279.618,A -85,B 0,C 180,E1 -6519.258,E2 -6519.258} C_VEL
LIN {X 0,Y 488.656,Z 279.614,A -85,B 0,C 180,E1 -6521.602,E2 -6521.602} C_VEL
LIN {X 0,Y 488.663,Z 279.61,A -85,B 0,C 180,E1 -6524.807,E2 -6524.807} C_VEL
LIN {X 0,Y 488.656,Z 279.617,A -85,B 0,C 180,E1 -6527.478,E2 -6527.478} C_VEL
LIN {X 0,Y 488.701,Z 279.613,A -85,B 0,C 180,E1 -6529.68,E2 -6529.68} C_VEL
LIN {X 0,Y 488.63,Z 279.613,A -85,B 0,C 180,E1 -6532.843,E2 -6532.843} C_VEL
LIN {X 0,Y 488.69,Z 279.612,A -85,B 0,C 180,E1 -6535.89,E2 -6535.89} C_VEL
LIN {X 0,Y 488.66,Z 279.612,A -85,B 0,C 180,E1 -6538.823,E2 -6538.823} C_VEL
LIN {X 0,Y 488.669,Z 279.612,A -85,B 0,C 180,E1 -6541.671,E2 -6541.671} C_VEL
LIN {X 0,Y 488.697,Z 279.775,A -85,B 0,C 180,E1 -6544.549,E2 -6544.549} C_VEL
LIN {X 0,Y 491.543,Z 293.056,A -85,B 0,C 180,E1 -6546.628,E2 -6546.628} C_VEL
LIN {X 0,Y 490.836,Z 311.527,A -85,B 0,C 180,E1 -6549.248,E2 -6549.248} C_VEL
LIN {X 0,Y 490.018,Z 333.08,A -85,B 0,C 180,E1 -6552.259,E2 -6552.259} C_VEL
LIN {X 0,Y 489.672,Z 345.106,A -85,B 0,C 180,E1 -6553.925,E2 -6553.925} C_VEL
LIN {X 0,Y 491.338,Z 358.274,A -85,B 0,C 180,E1 -6554.18,E2 -6554.18} C_VEL
LIN {X 0,Y 490.681,Z 452.223,A -85,B 0,C 180,E1 -6555.62,E2 -6555.62} C_VEL
LIN {X 0,Y 490.49,Z 461.775,A -85,B 0,C 180,E1 -6555.852,E2 -6555.852} C_VEL
LIN {X 0,Y 490.213,Z 472.197,A -85,B 0,C 180,E1 -6556.214,E2 -6556.214} C_VEL
LIN {X 0,Y 489.973,Z 481.358,A -85,B 0,C 180,E1 -6556.63,E2 -6556.63} C_VEL
LIN {X 0,Y 489.647,Z 492.065,A -85,B 0,C 180,E1 -6557.254,E2 -6557.254} C_VEL
LIN {X 0,Y 489.345,Z 502.113,A -85,B 0,C 180,E1 -6557.988,E2 -6557.988} C_VEL
LIN {X 0,Y 489.079,Z 510.381,A -85,B 0,C 180,E1 -6558.712,E2 -6558.712} C_VEL
LIN {X 0,Y 488.734,Z 519.239,A -85,B 0,C 180,E1 -6559.648,E2 -6559.648} C_VEL
LIN {X 0,Y 488.539,Z 525.936,A -85,B 0,C 180,E1 -6560.48,E2 -6560.48} C_VEL
LIN {X 0,Y 488.311,Z 532.932,A -85,B 0,C 180,E1 -6561.519,E2 -6561.519} C_VEL
LIN {X 0,Y 488.162,Z 538.775,A -85,B 0,C 180,E1 -6562.558,E2 -6562.558} C_VEL
LIN {X 0,Y 488.01,Z 544.418,A -85,B 0,C 180,E1 -6563.801,E2 -6563.801} C_VEL
LIN {X 0,Y 487.968,Z 548.86,A -85,B 0,C 180,E1 -6565.045,E2 -6565.045} C_VEL
LIN {X 0,Y 487.957,Z 551.193,A -85,B 0,C 180,E1 -6565.872,E2 -6565.872} C_VEL
LIN {X 0,Y 487.955,Z 554.551,A -85,B 0,C 180,E1 -6567.525,E2 -6567.525} C_VEL
LIN {X 0,Y 487.834,Z 556.099,A -85,B 0,C 180,E1 -6569.176,E2 -6569.176} C_VEL
LIN {X 0,Y 487.826,Z 556.385,A -85,B 0,C 180,E1 -6570.002,E2 -6570.002} C_VEL
LIN {X 0,Y 487.89,Z 555.474,A -85,B 0,C 180,E1 -6571.652,E2 -6571.652} C_VEL
LIN {X 0,Y 487.956,Z 554.48,A -85,B 0,C 180,E1 -6572.478,E2 -6572.478} C_VEL
LIN {X 0,Y 487.965,Z 551.075,A -85,B 0,C 180,E1 -6574.131,E2 -6574.131} C_VEL
LIN {X 0,Y 488.041,Z 547.335,A -85,B 0,C 180,E1 -6575.372,E2 -6575.372} C_VEL
LIN {X 0,Y 488.07,Z 542.435,A -85,B 0,C 180,E1 -6576.616,E2 -6576.616} C_VEL
LIN {X 0,Y 488.178,Z 537.423,A -85,B 0,C 180,E1 -6577.654,E2 -6577.654} C_VEL
LIN {X 0,Y 488.364,Z 529.921,A -85,B 0,C 180,E1 -6578.9,E2 -6578.9} C_VEL
LIN {X 0,Y 488.583,Z 522.306,A -85,B 0,C 180,E1 -6579.94,E2 -6579.94} C_VEL
LIN {X 0,Y 488.832,Z 514.066,A -85,B 0,C 180,E1 -6580.877,E2 -6580.877} C_VEL
LIN {X 0,Y 489.068,Z 506.523,A -85,B 0,C 180,E1 -6581.607,E2 -6581.607} C_VEL
LIN {X 0,Y 489.457,Z 496.013,A -85,B 0,C 180,E1 -6582.438,E2 -6582.438} C_VEL
LIN {X 0,Y 489.8,Z 486.325,A -85,B 0,C 180,E1 -6583.061,E2 -6583.061} C_VEL
LIN {X 0,Y 490.113,Z 476.225,A -85,B 0,C 180,E1 -6583.581,E2 -6583.581} C_VEL
LIN {X 0,Y 490.353,Z 465.707,A -85,B 0,C 180,E1 -6583.997,E2 -6583.997} C_VEL
LIN {X 0,Y 490.536,Z 454.571,A -85,B 0,C 180,E1 -6584.309,E2 -6584.309} C_VEL
LIN {X 0,Y 490.813,Z 435.995,A -85,B 0,C 180,E1 -6584.618,E2 -6584.618} C_VEL
LIN {X 0,Y 491.137,Z 356.743,A -85,B 0,C 180,E1 -6585.823,E2 -6585.823} C_VEL
LIN {X 0,Y 489.567,Z 344.756,A -85,B 0,C 180,E1 -6586.064,E2 -6586.064} C_VEL
LIN {X 0,Y 490.237,Z 320.798,A -85,B 0,C 180,E1 -6589.252,E2 -6589.252} C_VEL
LIN {X 0,Y 490.784,Z 299.559,A -85,B 0,C 180,E1 -6592.079,E2 -6592.079} C_VEL
LIN {X 0,Y 491.032,Z 291.695,A -85,B 0,C 180,E1 -6593.135,E2 -6593.135} C_VEL
LIN {X 0,Y 488.694,Z 279.614,A -85,B 0,C 180,E1 -6594.9,E2 -6594.9} C_VEL
LIN {X 0,Y 488.674,Z 279.621,A -85,B 0,C 180,E1 -6597.4,E2 -6597.4} C_VEL
LIN {X 0,Y 488.695,Z 279.611,A -85,B 0,C 180,E1 -6600.36,E2 -6600.36} C_VEL
LIN {X 0,Y 488.725,Z 279.611,A -85,B 0,C 180,E1 -6603.483,E2 -6603.483} C_VEL
LIN {X 0,Y 488.671,Z 279.611,A -85,B 0,C 180,E1 -6606.353,E2 -6606.353} C_VEL
LIN {X 0,Y 488.688,Z 279.613,A -85,B 0,C 180,E1 -6609.253,E2 -6609.253} C_VEL
LIN {X 0,Y 488.709,Z 279.613,A -85,B 0,C 180,E1 -6611.601,E2 -6611.601} C_VEL
LIN {X 0,Y 488.695,Z 279.608,A -85,B 0,C 180,E1 -6614.8,E2 -6614.8} C_VEL
LIN {X 0,Y 488.673,Z 279.613,A -85,B 0,C 180,E1 -6617.473,E2 -6617.473} C_VEL
LIN {X 0,Y 488.713,Z 279.609,A -85,B 0,C 180,E1 -6619.675,E2 -6619.675} C_VEL
LIN {X 0,Y 488.662,Z 279.614,A -85,B 0,C 180,E1 -6622.276,E2 -6622.276} C_VEL
LIN {X 0,Y 488.707,Z 279.602,A -85,B 0,C 180,E1 -6625.05,E2 -6625.05} C_VEL
LIN {X 0,Y 488.681,Z 279.61,A -85,B 0,C 180,E1 -6628.044,E2 -6628.044} C_VEL
LIN {X 0,Y 488.707,Z 279.606,A -85,B 0,C 180,E1 -6630.729,E2 -6630.729} C_VEL
LIN {X 0,Y 488.741,Z 279.6,A -85,B 0,C 180,E1 -6633.528,E2 -6633.528} C_VEL
LIN {X 0,Y 488.689,Z 279.613,A -85,B 0,C 180,E1 -6636.255,E2 -6636.255} C_VEL
LIN {X 0,Y 488.718,Z 279.606,A -85,B 0,C 180,E1 -6639.174,E2 -6639.174} C_VEL
LIN {X 0,Y 488.703,Z 279.612,A -85,B 0,C 180,E1 -6642.423,E2 -6642.423} C_VEL
LIN {X 0,Y 488.74,Z 279.607,A -85,B 0,C 180,E1 -6644.999,E2 -6644.999} C_VEL
LIN {X 0,Y 488.801,Z 279.597,A -85,B 0,C 180,E1 -6648.388,E2 -6648.388} C_VEL
LIN {X 0,Y 488.785,Z 279.601,A -85,B 0,C 180,E1 -6651.734,E2 -6651.734} C_VEL
LIN {X 0,Y 488.82,Z 279.596,A -85,B 0,C 180,E1 -6654.224,E2 -6654.224} C_VEL
LIN {X 0,Y 489.123,Z 279.641,A -85,B 0,C 180,E1 -6658.765,E2 -6658.765} C_VEL
LIN {X 0,Y 488.968,Z 299.38,A -85,B 0,C 180,E1 -6661.442,E2 -6661.442} C_VEL
LIN {X 0,Y 488.897,Z 321.2,A -85,B 0,C 180,E1 -6664.535,E2 -6664.535} C_VEL
LIN {X 0,Y 488.881,Z 337.804,A -85,B 0,C 180,E1 -6666.988,E2 -6666.988} C_VEL
LIN {X 0,Y 490.732,Z 350.397,A -85,B 0,C 180,E1 -6667.275,E2 -6667.275} C_VEL
LIN {X 0,Y 490.1,Z 419.562,A -85,B 0,C 180,E1 -6668.426,E2 -6668.426} C_VEL
LIN {X 0,Y 489.934,Z 430.453,A -85,B 0,C 180,E1 -6668.741,E2 -6668.741} C_VEL
LIN {X 0,Y 489.71,Z 440.825,A -85,B 0,C 180,E1 -6669.188,E2 -6669.188} C_VEL
LIN {X 0,Y 489.494,Z 451.361,A -85,B 0,C 180,E1 -6669.817,E2 -6669.817} C_VEL
LIN {X 0,Y 489.18,Z 459.758,A -85,B 0,C 180,E1 -6670.451,E2 -6670.451} C_VEL
LIN {X 0,Y 488.975,Z 466.65,A -85,B 0,C 180,E1 -6671.084,E2 -6671.084} C_VEL
LIN {X 0,Y 488.77,Z 474.367,A -85,B 0,C 180,E1 -6671.945,E2 -6671.945} C_VEL
LIN {X 0,Y 488.53,Z 481.238,A -85,B 0,C 180,E1 -6672.885,E2 -6672.885} C_VEL
LIN {X 0,Y 488.29,Z 488.522,A -85,B 0,C 180,E1 -6674.164,E2 -6674.164} C_VEL
LIN {X 0,Y 488.149,Z 493.407,A -85,B 0,C 180,E1 -6675.302,E2 -6675.302} C_VEL
LIN {X 0,Y 488.077,Z 496.723,A -85,B 0,C 180,E1 -6676.308,E2 -6676.308} C_VEL
LIN {X 0,Y 487.944,Z 499.752,A -85,B 0,C 180,E1 -6677.606,E2 -6677.606} C_VEL
LIN {X 0,Y 487.884,Z 501.015,A -85,B 0,C 180,E1 -6678.477,E2 -6678.477} C_VEL
LIN {X 0,Y 487.864,Z 501.733,A -85,B 0,C 180,E1 -6679.35,E2 -6679.35} C_VEL
LIN {X 0,Y 487.889,Z 501.766,A -85,B 0,C 180,E1 -6680.568,E2 -6680.568} C_VEL
LIN {X 0,Y 487.905,Z 501.513,A -85,B 0,C 180,E1 -6681.108,E2 -6681.108} C_VEL
LIN {X 0,Y 487.909,Z 500.472,A -85,B 0,C 180,E1 -6681.995,E2 -6681.995} C_VEL
LIN {X 0,Y 488.039,Z 497.821,A -85,B 0,C 180,E1 -6683.33,E2 -6683.33} C_VEL
LIN {X 0,Y 488.1,Z 495.235,A -85,B 0,C 180,E1 -6684.228,E2 -6684.228} C_VEL
LIN {X 0,Y 488.177,Z 491.573,A -85,B 0,C 180,E1 -6685.207,E2 -6685.207} C_VEL
LIN {X 0,Y 488.331,Z 486.479,A -85,B 0,C 180,E1 -6686.267,E2 -6686.267} C_VEL
LIN {X 0,Y 488.495,Z 480.635,A -85,B 0,C 180,E1 -6687.239,E2 -6687.239} C_VEL
LIN {X 0,Y 488.681,Z 474.329,A -85,B 0,C 180,E1 -6688.1,E2 -6688.1} C_VEL
LIN {X 0,Y 488.882,Z 466.732,A -85,B 0,C 180,E1 -6688.949,E2 -6688.949} C_VEL
LIN {X 0,Y 489.153,Z 458.293,A -85,B 0,C 180,E1 -6689.715,E2 -6689.715} C_VEL
LIN {X 0,Y 489.433,Z 448.575,A -85,B 0,C 180,E1 -6690.421,E2 -6690.421} C_VEL
LIN {X 0,Y 489.721,Z 437.619,A -85,B 0,C 180,E1 -6691.012,E2 -6691.012} C_VEL
LIN {X 0,Y 489.889,Z 427.877,A -85,B 0,C 180,E1 -6691.396,E2 -6691.396} C_VEL
LIN {X 0,Y 490.01,Z 418.185,A -85,B 0,C 180,E1 -6691.659,E2 -6691.659} C_VEL
LIN {X 0,Y 490.527,Z 349.802,A -85,B 0,C 180,E1 -6692.761,E2 -6692.761} C_VEL
LIN {X 0,Y 488.856,Z 338.796,A -85,B 0,C 180,E1 -6693.003,E2 -6693.003} C_VEL
LIN {X 0,Y 489.314,Z 319.682,A -85,B 0,C 180,E1 -6696.46,E2 -6696.46} C_VEL
LIN {X 0,Y 489.63,Z 309.134,A -85,B 0,C 180,E1 -6698.389,E2 -6698.389} C_VEL
LIN {X 0,Y 489.011,Z 306.082,A -85,B 0,C 180,E1 -6698.977,E2 -6698.977} C_VEL
LIN {X 0,Y 483.621,Z 296.771,A -85,B 0,C 180,E1 -6700.946,E2 -6700.946} C_VEL
LIN {X 0,Y 483.088,Z 293.73,A -85,B 0,C 180,E1 -6701.546,E2 -6701.546} C_VEL
LIN {X 0,Y 483.022,Z 287.582,A -85,B 0,C 180,E1 -6702.716,E2 -6702.716} C_VEL
LIN {X 0,Y 481.66,Z 280.489,A -85,B 0,C 180,E1 -6704.176,E2 -6704.176} C_VEL
LIN {X 0,Y 481.621,Z 280.492,A -85,B 0,C 180,E1 -6706.855,E2 -6706.855} C_VEL
LIN {X 0,Y 481.666,Z 280.482,A -85,B 0,C 180,E1 -6710.061,E2 -6710.061} C_VEL
LIN {X 0,Y 481.611,Z 280.493,A -85,B 0,C 180,E1 -6713.38,E2 -6713.38} C_VEL
LIN {X 0,Y 481.666,Z 280.483,A -85,B 0,C 180,E1 -6716.328,E2 -6716.328} C_VEL
LIN {X 0,Y 481.642,Z 280.485,A -85,B 0,C 180,E1 -6719.42,E2 -6719.42} C_VEL
LIN {X 0,Y 481.648,Z 280.492,A -85,B 0,C 180,E1 -6722.166,E2 -6722.166} C_VEL
LIN {X 0,Y 481.673,Z 280.481,A -85,B 0,C 180,E1 -6724.968,E2 -6724.968} C_VEL
LIN {X 0,Y 481.637,Z 280.485,A -85,B 0,C 180,E1 -6727.705,E2 -6727.705} C_VEL
LIN {X 0,Y 481.698,Z 280.483,A -85,B 0,C 180,E1 -6730.393,E2 -6730.393} C_VEL
LIN {X 0,Y 481.669,Z 280.485,A -85,B 0,C 180,E1 -6733.033,E2 -6733.033} C_VEL
LIN {X 0,Y 481.674,Z 280.48,A -85,B 0,C 180,E1 -6735.638,E2 -6735.638} C_VEL
LIN {X 0,Y 481.755,Z 280.47,A -85,B 0,C 180,E1 -6738.215,E2 -6738.215} C_VEL
LIN {X 0,Y 481.721,Z 280.478,A -85,B 0,C 180,E1 -6741.61,E2 -6741.61} C_VEL
LIN {X 0,Y 481.777,Z 280.467,A -85,B 0,C 180,E1 -6744.138,E2 -6744.138} C_VEL
LIN {X 0,Y 481.908,Z 280.459,A -85,B 0,C 180,E1 -6747.491,E2 -6747.491} C_VEL
LIN {X 0,Y 481.913,Z 280.455,A -85,B 0,C 180,E1 -6749.998,E2 -6749.998} C_VEL
LIN {X 0,Y 481.908,Z 280.452,A -85,B 0,C 180,E1 -6752.506,E2 -6752.506} C_VEL
LIN {X 0,Y 481.774,Z 280.473,A -85,B 0,C 180,E1 -6755.859,E2 -6755.859} C_VEL
LIN {X 0,Y 481.717,Z 280.481,A -85,B 0,C 180,E1 -6758.387,E2 -6758.387} C_VEL
LIN {X 0,Y 481.749,Z 280.471,A -85,B 0,C 180,E1 -6761.782,E2 -6761.782} C_VEL
LIN {X 0,Y 481.736,Z 280.473,A -85,B 0,C 180,E1 -6765.221,E2 -6765.221} C_VEL
LIN {X 0,Y 481.7,Z 280.485,A -85,B 0,C 180,E1 -6768.718,E2 -6768.718} C_VEL
LIN {X 0,Y 481.636,Z 280.487,A -85,B 0,C 180,E1 -6771.391,E2 -6771.391} C_VEL
LIN {X 0,Y 481.637,Z 280.484,A -85,B 0,C 180,E1 -6774.111,E2 -6774.111} C_VEL
LIN {X 0,Y 481.663,Z 280.488,A -85,B 0,C 180,E1 -6777.118,E2 -6777.118} C_VEL
LIN {X 0,Y 481.656,Z 280.487,A -85,B 0,C 180,E1 -6779.737,E2 -6779.737} C_VEL
LIN {X 0,Y 481.653,Z 280.482,A -85,B 0,C 180,E1 -6782.67,E2 -6782.67} C_VEL
LIN {X 0,Y 481.615,Z 280.495,A -85,B 0,C 180,E1 -6785.705,E2 -6785.705} C_VEL
LIN {X 0,Y 481.644,Z 280.483,A -85,B 0,C 180,E1 -6788.855,E2 -6788.855} C_VEL
LIN {X 0,Y 481.624,Z 280.492,A -85,B 0,C 180,E1 -6791.908,E2 -6791.908} C_VEL
LIN {X 0,Y 481.623,Z 280.493,A -85,B 0,C 180,E1 -6794.454,E2 -6794.454} C_VEL
LIN {X 0,Y 481.613,Z 280.488,A -85,B 0,C 180,E1 -6797.835,E2 -6797.835} C_VEL
LIN {X 0,Y 481.642,Z 280.493,A -85,B 0,C 180,E1 -6800.647,E2 -6800.647} C_VEL
LIN {X 0,Y 481.589,Z 280.492,A -85,B 0,C 180,E1 -6803.372,E2 -6803.372} C_VEL
LIN {X 0,Y 481.627,Z 280.487,A -85,B 0,C 180,E1 -6806.323,E2 -6806.323} C_VEL
LIN {X 0,Y 481.611,Z 280.493,A -85,B 0,C 180,E1 -6809.413,E2 -6809.413} C_VEL
LIN {X 0,Y 481.655,Z 280.482,A -85,B 0,C 180,E1 -6812.165,E2 -6812.165} C_VEL
LIN {X 0,Y 481.668,Z 280.483,A -85,B 0,C 180,E1 -6814.967,E2 -6814.967} C_VEL
LIN {X 0,Y 481.606,Z 280.496,A -85,B 0,C 180,E1 -6817.702,E2 -6817.702} C_VEL
LIN {X 0,Y 481.65,Z 280.484,A -85,B 0,C 180,E1 -6820.39,E2 -6820.39} C_VEL
LIN {X 0,Y 481.635,Z 280.484,A -85,B 0,C 180,E1 -6823.031,E2 -6823.031} C_VEL
LIN {X 0,Y 481.638,Z 280.487,A -85,B 0,C 180,E1 -6825.637,E2 -6825.637} C_VEL
LIN {X 0,Y 481.735,Z 280.482,A -85,B 0,C 180,E1 -6828.214,E2 -6828.214} C_VEL
LIN {X 0,Y 481.703,Z 280.476,A -85,B 0,C 180,E1 -6831.61,E2 -6831.61} C_VEL
LIN {X 0,Y 481.771,Z 280.471,A -85,B 0,C 180,E1 -6834.139,E2 -6834.139} C_VEL
LIN {X 0,Y 481.872,Z 280.455,A -85,B 0,C 180,E1 -6837.492,E2 -6837.492} C_VEL
LIN {X 0,Y 481.874,Z 280.455,A -85,B 0,C 180,E1 -6840,E2 -6840} C_VEL
LIN {X 0,Y 481.872,Z 280.457,A -85,B 0,C 180,E1 -6842.507,E2 -6842.507} C_VEL
LIN {X 0,Y 481.77,Z 280.469,A -85,B 0,C 180,E1 -6845.861,E2 -6845.861} C_VEL
LIN {X 0,Y 481.702,Z 280.476,A -85,B 0,C 180,E1 -6848.389,E2 -6848.389} C_VEL
LIN {X 0,Y 481.734,Z 280.478,A -85,B 0,C 180,E1 -6851.785,E2 -6851.785} C_VEL
LIN {X 0,Y 481.685,Z 280.48,A -85,B 0,C 180,E1 -6855.226,E2 -6855.226} C_VEL
LIN {X 0,Y 481.654,Z 280.482,A -85,B 0,C 180,E1 -6858.724,E2 -6858.724} C_VEL
LIN {X 0,Y 481.602,Z 280.489,A -85,B 0,C 180,E1 -6861.396,E2 -6861.396} C_VEL
LIN {X 0,Y 481.629,Z 280.492,A -85,B 0,C 180,E1 -6864.115,E2 -6864.115} C_VEL
LIN {X 0,Y 481.694,Z 280.478,A -85,B 0,C 180,E1 -6867.142,E2 -6867.142} C_VEL
LIN {X 0,Y 481.627,Z 280.485,A -85,B 0,C 180,E1 -6869.744,E2 -6869.744} C_VEL
LIN {X 0,Y 481.623,Z 280.494,A -85,B 0,C 180,E1 -6872.677,E2 -6872.677} C_VEL
LIN {X 0,Y 481.595,Z 280.49,A -85,B 0,C 180,E1 -6875.713,E2 -6875.713} C_VEL
LIN {X 0,Y 481.627,Z 280.491,A -85,B 0,C 180,E1 -6878.863,E2 -6878.863} C_VEL
LIN {X 0,Y 481.606,Z 280.489,A -85,B 0,C 180,E1 -6881.915,E2 -6881.915} C_VEL
LIN {X 0,Y 481.616,Z 280.487,A -85,B 0,C 180,E1 -6884.462,E2 -6884.462} C_VEL
LIN {X 0,Y 481.613,Z 280.493,A -85,B 0,C 180,E1 -6887.843,E2 -6887.843} C_VEL
LIN {X 0,Y 481.62,Z 280.486,A -85,B 0,C 180,E1 -6890.659,E2 -6890.659} C_VEL
LIN {X 0,Y 481.588,Z 280.492,A -85,B 0,C 180,E1 -6893.382,E2 -6893.382} C_VEL
LIN {X 0,Y 481.644,Z 280.489,A -85,B 0,C 180,E1 -6896.331,E2 -6896.331} C_VEL
LIN {X 0,Y 481.618,Z 280.487,A -85,B 0,C 180,E1 -6899.423,E2 -6899.423} C_VEL
LIN {X 0,Y 481.626,Z 280.493,A -85,B 0,C 180,E1 -6902.168,E2 -6902.168} C_VEL
LIN {X 0,Y 481.647,Z 280.573,A -85,B 0,C 180,E1 -6904.303,E2 -6904.303} C_VEL
LIN {X 0,Y 484.654,Z 294.66,A -85,B 0,C 180,E1 -6906.544,E2 -6906.544} C_VEL
LIN {X 0,Y 483.799,Z 314.378,A -85,B 0,C 180,E1 -6909.378,E2 -6909.378} C_VEL
LIN {X 0,Y 483.03,Z 334.382,A -85,B 0,C 180,E1 -6912.213,E2 -6912.213} C_VEL
LIN {X 0,Y 482.697,Z 345.357,A -85,B 0,C 180,E1 -6913.72,E2 -6913.72} C_VEL
LIN {X 0,Y 484.449,Z 359.951,A -85,B 0,C 180,E1 -6914.003,E2 -6914.003} C_VEL
LIN {X 0,Y 483.76,Z 451.759,A -85,B 0,C 180,E1 -6915.436,E2 -6915.436} C_VEL
LIN {X 0,Y 483.568,Z 461.38,A -85,B 0,C 180,E1 -6915.672,E2 -6915.672} C_VEL
LIN {X 0,Y 483.274,Z 471.221,A -85,B 0,C 180,E1 -6916.012,E2 -6916.012} C_VEL
LIN {X 0,Y 483.027,Z 480.537,A -85,B 0,C 180,E1 -6916.434,E2 -6916.434} C_VEL
LIN {X 0,Y 482.646,Z 491.928,A -85,B 0,C 180,E1 -6917.108,E2 -6917.108} C_VEL
LIN {X 0,Y 482.41,Z 500.322,A -85,B 0,C 180,E1 -6917.714,E2 -6917.714} C_VEL
LIN {X 0,Y 482.077,Z 509.792,A -85,B 0,C 180,E1 -6918.546,E2 -6918.546} C_VEL
LIN {X 0,Y 481.702,Z 518.692,A -85,B 0,C 180,E1 -6919.495,E2 -6919.495} C_VEL
LIN {X 0,Y 481.431,Z 526.859,A -85,B 0,C 180,E1 -6920.55,E2 -6920.55} C_VEL
LIN {X 0,Y 481.196,Z 533.64,A -85,B 0,C 180,E1 -6921.604,E2 -6921.604} C_VEL
LIN {X 0,Y 481.069,Z 538.317,A -85,B 0,C 180,E1 -6922.447,E2 -6922.447} C_VEL
LIN {X 0,Y 480.911,Z 544.441,A -85,B 0,C 180,E1 -6923.833,E2 -6923.833} C_VEL
LIN {X 0,Y 480.901,Z 548.446,A -85,B 0,C 180,E1 -6924.972,E2 -6924.972} C_VEL
LIN {X 0,Y 480.855,Z 550.778,A -85,B 0,C 180,E1 -6925.811,E2 -6925.811} C_VEL
LIN {X 0,Y 480.865,Z 554.153,A -85,B 0,C 180,E1 -6927.489,E2 -6927.489} C_VEL
LIN {X 0,Y 480.76,Z 555.705,A -85,B 0,C 180,E1 -6929.164,E2 -6929.164} C_VEL
LIN {X 0,Y 480.75,Z 555.991,A -85,B 0,C 180,E1 -6930.002,E2 -6930.002} C_VEL
LIN {X 0,Y 480.821,Z 555.075,A -85,B 0,C 180,E1 -6931.677,E2 -6931.677} C_VEL
LIN {X 0,Y 480.866,Z 554.077,A -85,B 0,C 180,E1 -6932.514,E2 -6932.514} C_VEL
LIN {X 0,Y 480.863,Z 550.659,A -85,B 0,C 180,E1 -6934.192,E2 -6934.192} C_VEL
LIN {X 0,Y 480.946,Z 546.908,A -85,B 0,C 180,E1 -6935.452,E2 -6935.452} C_VEL
LIN {X 0,Y 480.999,Z 541.994,A -85,B 0,C 180,E1 -6936.714,E2 -6936.714} C_VEL
LIN {X 0,Y 481.09,Z 536.961,A -85,B 0,C 180,E1 -6937.767,E2 -6937.767} C_VEL
LIN {X 0,Y 481.307,Z 529.436,A -85,B 0,C 180,E1 -6939.032,E2 -6939.032} C_VEL
LIN {X 0,Y 481.551,Z 521.791,A -85,B 0,C 180,E1 -6940.087,E2 -6940.087} C_VEL
LIN {X 0,Y 481.775,Z 514.549,A -85,B 0,C 180,E1 -6940.932,E2 -6940.932} C_VEL
LIN {X 0,Y 482.066,Z 505.924,A -85,B 0,C 180,E1 -6941.778,E2 -6941.778} C_VEL
LIN {X 0,Y 482.455,Z 495.945,A -85,B 0,C 180,E1 -6942.58,E2 -6942.58} C_VEL
LIN {X 0,Y 482.786,Z 487.467,A -85,B 0,C 180,E1 -6943.148,E2 -6943.148} C_VEL
LIN {X 0,Y 483.134,Z 476.571,A -85,B 0,C 180,E1 -6943.727,E2 -6943.727} C_VEL
LIN {X 0,Y 483.418,Z 465.459,A -85,B 0,C 180,E1 -6944.175,E2 -6944.175} C_VEL
LIN {X 0,Y 483.616,Z 454.354,A -85,B 0,C 180,E1 -6944.491,E2 -6944.491} C_VEL
LIN {X 0,Y 483.924,Z 434.193,A -85,B 0,C 180,E1 -6944.831,E2 -6944.831} C_VEL
LIN {X 0,Y 484.385,Z 358.295,A -85,B 0,C 180,E1 -6946.008,E2 -6946.008} C_VEL
LIN {X 0,Y 482.597,Z 344.579,A -85,B 0,C 180,E1 -6946.302,E2 -6946.302} C_VEL
LIN {X 0,Y 483.316,Z 320.511,A -85,B 0,C 180,E1 -6949.539,E2 -6949.539} C_VEL
LIN {X 0,Y 483.891,Z 300.992,A -85,B 0,C 180,E1 -6952.186,E2 -6952.186} C_VEL
LIN {X 0,Y 483.994,Z 292.078,A -85,B 0,C 180,E1 -6953.4,E2 -6953.4} C_VEL
LIN {X 0,Y 481.667,Z 280.49,A -85,B 0,C 180,E1 -6955.131,E2 -6955.131} C_VEL
LIN {X 0,Y 481.64,Z 280.495,A -85,B 0,C 180,E1 -6957.835,E2 -6957.835} C_VEL
LIN {X 0,Y 481.632,Z 280.492,A -85,B 0,C 180,E1 -6960.71,E2 -6960.71} C_VEL
LIN {X 0,Y 481.688,Z 280.486,A -85,B 0,C 180,E1 -6963.732,E2 -6963.732} C_VEL
LIN {X 0,Y 481.614,Z 280.49,A -85,B 0,C 180,E1 -6966.746,E2 -6966.746} C_VEL
LIN {X 0,Y 481.663,Z 280.491,A -85,B 0,C 180,E1 -6969.939,E2 -6969.939} C_VEL
LIN {X 0,Y 481.65,Z 280.489,A -85,B 0,C 180,E1 -6973.295,E2 -6973.295} C_VEL
LIN {X 0,Y 481.641,Z 280.492,A -85,B 0,C 180,E1 -6975.639,E2 -6975.639} C_VEL
LIN {X 0,Y 481.649,Z 280.485,A -85,B 0,C 180,E1 -6978.958,E2 -6978.958} C_VEL
LIN {X 0,Y 481.677,Z 280.481,A -85,B 0,C 180,E1 -6981.142,E2 -6981.142} C_VEL
LIN {X 0,Y 481.647,Z 280.482,A -85,B 0,C 180,E1 -6984.793,E2 -6984.793} C_VEL
LIN {X 0,Y 481.649,Z 280.479,A -85,B 0,C 180,E1 -6987.325,E2 -6987.325} C_VEL
LIN {X 0,Y 481.662,Z 280.486,A -85,B 0,C 180,E1 -6990.258,E2 -6990.258} C_VEL
LIN {X 0,Y 481.725,Z 280.474,A -85,B 0,C 180,E1 -6993.111,E2 -6993.111} C_VEL
LIN {X 0,Y 481.667,Z 280.484,A -85,B 0,C 180,E1 -6995.887,E2 -6995.887} C_VEL
LIN {X 0,Y 481.682,Z 280.484,A -85,B 0,C 180,E1 -6999.024,E2 -6999.024} C_VEL
LIN {X 0,Y 481.676,Z 280.484,A -85,B 0,C 180,E1 -7002.158,E2 -7002.158} C_VEL
LIN {X 0,Y 481.718,Z 280.483,A -85,B 0,C 180,E1 -7004.775,E2 -7004.775} C_VEL
LIN {X 0,Y 481.765,Z 280.472,A -85,B 0,C 180,E1 -7008.216,E2 -7008.216} C_VEL
LIN {X 0,Y 481.731,Z 280.48,A -85,B 0,C 180,E1 -7011.612,E2 -7011.612} C_VEL
LIN {X 0,Y 481.779,Z 280.474,A -85,B 0,C 180,E1 -7014.14,E2 -7014.14} C_VEL
LIN {X 0,Y 482.095,Z 280.48,A -85,B 0,C 180,E1 -7018.617,E2 -7018.617} C_VEL
LIN {X 0,Y 482.019,Z 299.734,A -85,B 0,C 180,E1 -7021.254,E2 -7021.254} C_VEL
LIN {X 0,Y 481.928,Z 321.781,A -85,B 0,C 180,E1 -7024.391,E2 -7024.391} C_VEL
LIN {X 0,Y 481.953,Z 338.161,A -85,B 0,C 180,E1 -7026.777,E2 -7026.777} C_VEL
LIN {X 0,Y 483.863,Z 350.802,A -85,B 0,C 180,E1 -7027.06,E2 -7027.06} C_VEL
LIN {X 0,Y 483.19,Z 419.491,A -85,B 0,C 180,E1 -7028.239,E2 -7028.239} C_VEL
LIN {X 0,Y 482.982,Z 429.736,A -85,B 0,C 180,E1 -7028.533,E2 -7028.533} C_VEL
LIN {X 0,Y 482.755,Z 441.479,A -85,B 0,C 180,E1 -7029.041,E2 -7029.041} C_VEL
LIN {X 0,Y 482.536,Z 451.416,A -85,B 0,C 180,E1 -7029.643,E2 -7029.643} C_VEL
LIN {X 0,Y 482.219,Z 459.861,A -85,B 0,C 180,E1 -7030.285,E2 -7030.285} C_VEL
LIN {X 0,Y 481.972,Z 467.839,A -85,B 0,C 180,E1 -7031.034,E2 -7031.034} C_VEL
LIN {X 0,Y 481.763,Z 474.438,A -85,B 0,C 180,E1 -7031.785,E2 -7031.785} C_VEL
LIN {X 0,Y 481.524,Z 480.74,A -85,B 0,C 180,E1 -7032.647,E2 -7032.647} C_VEL
LIN {X 0,Y 481.291,Z 487.178,A -85,B 0,C 180,E1 -7033.727,E2 -7033.727} C_VEL
LIN {X 0,Y 481.148,Z 492.252,A -85,B 0,C 180,E1 -7034.811,E2 -7034.811} C_VEL
LIN {X 0,Y 481.036,Z 496.757,A -85,B 0,C 180,E1 -7036.117,E2 -7036.117} C_VEL
LIN {X 0,Y 480.911,Z 499.054,A -85,B 0,C 180,E1 -7036.995,E2 -7036.995} C_VEL
LIN {X 0,Y 480.84,Z 501.131,A -85,B 0,C 180,E1 -7038.199,E2 -7038.199} C_VEL
LIN {X 0,Y 480.8,Z 501.764,A -85,B 0,C 180,E1 -7038.759,E2 -7038.759} C_VEL
LIN {X 0,Y 480.775,Z 502.243,A -85,B 0,C 180,E1 -7039.647,E2 -7039.647} C_VEL
LIN {X 0,Y 480.818,Z 502.105,A -85,B 0,C 180,E1 -7040.706,E2 -7040.706} C_VEL
LIN {X 0,Y 480.818,Z 501.56,A -85,B 0,C 180,E1 -7041.434,E2 -7041.434} C_VEL
LIN {X 0,Y 480.843,Z 500.37,A -85,B 0,C 180,E1 -7042.335,E2 -7042.335} C_VEL
LIN {X 0,Y 480.947,Z 498.548,A -85,B 0,C 180,E1 -7043.238,E2 -7043.238} C_VEL
LIN {X 0,Y 481.037,Z 494.442,A -85,B 0,C 180,E1 -7044.607,E2 -7044.607} C_VEL
LIN {X 0,Y 481.191,Z 489.751,A -85,B 0,C 180,E1 -7045.755,E2 -7045.755} C_VEL
LIN {X 0,Y 481.341,Z 484.989,A -85,B 0,C 180,E1 -7046.679,E2 -7046.679} C_VEL
LIN {X 0,Y 481.487,Z 478.993,A -85,B 0,C 180,E1 -7047.63,E2 -7047.63} C_VEL
LIN {X 0,Y 481.805,Z 471.008,A -85,B 0,C 180,E1 -7048.656,E2 -7048.656} C_VEL
LIN {X 0,Y 482.105,Z 461.63,A -85,B 0,C 180,E1 -7049.593,E2 -7049.593} C_VEL
LIN {X 0,Y 482.381,Z 452.749,A -85,B 0,C 180,E1 -7050.296,E2 -7050.296} C_VEL
LIN {X 0,Y 482.61,Z 444.151,A -85,B 0,C 180,E1 -7050.842,E2 -7050.842} C_VEL
LIN {X 0,Y 482.786,Z 435.961,A -85,B 0,C 180,E1 -7051.253,E2 -7051.253} C_VEL
LIN {X 0,Y 482.96,Z 426.13,A -85,B 0,C 180,E1 -7051.623,E2 -7051.623} C_VEL
LIN {X 0,Y 483.074,Z 415.416,A -85,B 0,C 180,E1 -7051.891,E2 -7051.891} C_VEL
LIN {X 0,Y 483.625,Z 350.546,A -85,B 0,C 180,E1 -7052.946,E2 -7052.946} C_VEL
LIN {X 0,Y 481.81,Z 338.797,A -85,B 0,C 180,E1 -7053.217,E2 -7053.217} C_VEL
LIN {X 0,Y 482.35,Z 319.814,A -85,B 0,C 180,E1 -7056.683,E2 -7056.683} C_VEL
LIN {X 0,Y 482.772,Z 304.569,A -85,B 0,C 180,E1 -7059.511,E2 -7059.511} C_VEL
LIN {X 0,Y 483.088,Z 293.73,A -85,B 0,C 180,E1 -7061.546,E2 -7061.546} C_VEL
LIN {X 0,Y 482.454,Z 291.778,A -85,B 0,C 180,E1 -7061.944,E2 -7061.944} C_VEL
LIN {X 0,Y 479.523,Z 289.119,A -85,B 0,C 180,E1 -7062.587,E2 -7062.587} C_VEL
LIN {X 0,Y 476.302,Z 286.534,A -85,B 0,C 180,E1 -7063.239,E2 -7063.239} C_VEL
LIN {X 0,Y 475.255,Z 284.67,A -85,B 0,C 180,E1 -7063.652,E2 -7063.652} C_VEL
LIN {X 0,Y 474.601,Z 281.369,A -85,B 0,C 180,E1 -7064.376,E2 -7064.376} C_VEL
LIN {X 0,Y 474.614,Z 281.363,A -85,B 0,C 180,E1 -7067.765,E2 -7067.765} C_VEL
LIN {X 0,Y 474.619,Z 281.358,A -85,B 0,C 180,E1 -7070.454,E2 -7070.454} C_VEL
LIN {X 0,Y 474.574,Z 281.373,A -85,B 0,C 180,E1 -7073.677,E2 -7073.677} C_VEL
LIN {X 0,Y 474.611,Z 281.359,A -85,B 0,C 180,E1 -7076.779,E2 -7076.779} C_VEL
LIN {X 0,Y 474.594,Z 281.367,A -85,B 0,C 180,E1 -7079.77,E2 -7079.77} C_VEL
LIN {X 0,Y 474.601,Z 281.363,A -85,B 0,C 180,E1 -7082.686,E2 -7082.686} C_VEL
LIN {X 0,Y 474.625,Z 281.358,A -85,B 0,C 180,E1 -7085.506,E2 -7085.506} C_VEL
LIN {X 0,Y 474.659,Z 281.355,A -85,B 0,C 180,E1 -7089.185,E2 -7089.185} C_VEL
LIN {X 0,Y 474.646,Z 281.355,A -85,B 0,C 180,E1 -7091.884,E2 -7091.884} C_VEL
LIN {X 0,Y 474.701,Z 281.353,A -85,B 0,C 180,E1 -7094.544,E2 -7094.544} C_VEL
LIN {X 0,Y 474.709,Z 281.347,A -85,B 0,C 180,E1 -7098.037,E2 -7098.037} C_VEL
LIN {X 0,Y 474.67,Z 281.358,A -85,B 0,C 180,E1 -7101.485,E2 -7101.485} C_VEL
LIN {X 0,Y 474.741,Z 281.344,A -85,B 0,C 180,E1 -7104.051,E2 -7104.051} C_VEL
LIN {X 0,Y 474.873,Z 281.334,A -85,B 0,C 180,E1 -7107.454,E2 -7107.454} C_VEL
LIN {X 0,Y 474.883,Z 281.331,A -85,B 0,C 180,E1 -7109.998,E2 -7109.998} C_VEL
LIN {X 0,Y 474.873,Z 281.328,A -85,B 0,C 180,E1 -7112.543,E2 -7112.543} C_VEL
LIN {X 0,Y 474.737,Z 281.351,A -85,B 0,C 180,E1 -7115.946,E2 -7115.946} C_VEL
LIN {X 0,Y 474.666,Z 281.357,A -85,B 0,C 180,E1 -7118.512,E2 -7118.512} C_VEL
LIN {X 0,Y 474.703,Z 281.351,A -85,B 0,C 180,E1 -7121.959,E2 -7121.959} C_VEL
LIN {X 0,Y 474.677,Z 281.351,A -85,B 0,C 180,E1 -7125.764,E2 -7125.764} C_VEL
LIN {X 0,Y 474.654,Z 281.361,A -85,B 0,C 180,E1 -7129.007,E2 -7129.007} C_VEL
LIN {X 0,Y 474.579,Z 281.364,A -85,B 0,C 180,E1 -7131.725,E2 -7131.725} C_VEL
LIN {X 0,Y 474.615,Z 281.36,A -85,B 0,C 180,E1 -7134.491,E2 -7134.491} C_VEL
LIN {X 0,Y 474.624,Z 281.367,A -85,B 0,C 180,E1 -7137.32,E2 -7137.32} C_VEL
LIN {X 0,Y 474.585,Z 281.363,A -85,B 0,C 180,E1 -7140.226,E2 -7140.226} C_VEL
LIN {X 0,Y 474.624,Z 281.361,A -85,B 0,C 180,E1 -7143.216,E2 -7143.216} C_VEL
LIN {X 0,Y 474.567,Z 281.367,A -85,B 0,C 180,E1 -7146.319,E2 -7146.319} C_VEL
LIN {X 0,Y 474.591,Z 281.366,A -85,B 0,C 180,E1 -7149.641,E2 -7149.641} C_VEL
LIN {X 0,Y 474.595,Z 281.37,A -85,B 0,C 180,E1 -7152.232,E2 -7152.232} C_VEL
LIN {X 0,Y 474.585,Z 281.363,A -85,B 0,C 180,E1 -7155.293,E2 -7155.293} C_VEL
LIN {X 0,Y 474.586,Z 281.367,A -85,B 0,C 180,E1 -7158.21,E2 -7158.21} C_VEL
LIN {X 0,Y 474.607,Z 281.367,A -85,B 0,C 180,E1 -7160.45,E2 -7160.45} C_VEL
LIN {X 0,Y 474.551,Z 281.367,A -85,B 0,C 180,E1 -7163.672,E2 -7163.672} C_VEL
LIN {X 0,Y 474.571,Z 281.371,A -85,B 0,C 180,E1 -7166.774,E2 -7166.774} C_VEL
LIN {X 0,Y 474.566,Z 281.366,A -85,B 0,C 180,E1 -7169.767,E2 -7169.767} C_VEL
LIN {X 0,Y 474.65,Z 281.356,A -85,B 0,C 180,E1 -7172.676,E2 -7172.676} C_VEL
LIN {X 0,Y 474.61,Z 281.369,A -85,B 0,C 180,E1 -7175.504,E2 -7175.504} C_VEL
LIN {X 0,Y 474.617,Z 281.361,A -85,B 0,C 180,E1 -7179.182,E2 -7179.182} C_VEL
LIN {X 0,Y 474.601,Z 281.37,A -85,B 0,C 180,E1 -7181.882,E2 -7181.882} C_VEL
LIN {X 0,Y 474.643,Z 281.357,A -85,B 0,C 180,E1 -7184.542,E2 -7184.542} C_VEL
LIN {X 0,Y 474.679,Z 281.358,A -85,B 0,C 180,E1 -7188.036,E2 -7188.036} C_VEL
LIN {X 0,Y 474.669,Z 281.352,A -85,B 0,C 180,E1 -7191.485,E2 -7191.485} C_VEL
LIN {X 0,Y 474.731,Z 281.347,A -85,B 0,C 180,E1 -7194.051,E2 -7194.051} C_VEL
LIN {X 0,Y 474.84,Z 281.332,A -85,B 0,C 180,E1 -7197.455,E2 -7197.455} C_VEL
LIN {X 0,Y 474.817,Z 281.342,A -85,B 0,C 180,E1 -7200.848,E2 -7200.848} C_VEL
LIN {X 0,Y 474.839,Z 281.333,A -85,B 0,C 180,E1 -7202.544,E2 -7202.544} C_VEL
LIN {X 0,Y 474.73,Z 281.345,A -85,B 0,C 180,E1 -7205.948,E2 -7205.948} C_VEL
LIN {X 0,Y 474.668,Z 281.352,A -85,B 0,C 180,E1 -7208.514,E2 -7208.514} C_VEL
LIN {X 0,Y 474.677,Z 281.355,A -85,B 0,C 180,E1 -7211.963,E2 -7211.963} C_VEL
LIN {X 0,Y 474.641,Z 281.36,A -85,B 0,C 180,E1 -7215.457,E2 -7215.457} C_VEL
LIN {X 0,Y 474.607,Z 281.36,A -85,B 0,C 180,E1 -7219.012,E2 -7219.012} C_VEL
LIN {X 0,Y 474.55,Z 281.37,A -85,B 0,C 180,E1 -7221.73,E2 -7221.73} C_VEL
LIN {X 0,Y 474.608,Z 281.366,A -85,B 0,C 180,E1 -7224.495,E2 -7224.495} C_VEL
LIN {X 0,Y 474.629,Z 281.357,A -85,B 0,C 180,E1 -7227.337,E2 -7227.337} C_VEL
LIN {X 0,Y 474.553,Z 281.374,A -85,B 0,C 180,E1 -7230.813,E2 -7230.813} C_VEL
LIN {X 0,Y 474.591,Z 281.362,A -85,B 0,C 180,E1 -7233.987,E2 -7233.987} C_VEL
LIN {X 0,Y 474.529,Z 281.378,A -85,B 0,C 180,E1 -7236.903,E2 -7236.903} C_VEL
LIN {X 0,Y 474.565,Z 281.368,A -85,B 0,C 180,E1 -7239.648,E2 -7239.648} C_VEL
LIN {X 0,Y 474.56,Z 281.366,A -85,B 0,C 180,E1 -7242.237,E2 -7242.237} C_VEL
LIN {X 0,Y 474.58,Z 281.37,A -85,B 0,C 180,E1 -7245.302,E2 -7245.302} C_VEL
LIN {X 0,Y 474.586,Z 281.364,A -85,B 0,C 180,E1 -7248.218,E2 -7248.218} C_VEL
LIN {X 0,Y 474.595,Z 281.362,A -85,B 0,C 180,E1 -7250.456,E2 -7250.456} C_VEL
LIN {X 0,Y 474.551,Z 281.372,A -85,B 0,C 180,E1 -7253.679,E2 -7253.679} C_VEL
LIN {X 0,Y 474.588,Z 281.363,A -85,B 0,C 180,E1 -7256.781,E2 -7256.781} C_VEL
LIN {X 0,Y 474.57,Z 281.367,A -85,B 0,C 180,E1 -7259.773,E2 -7259.773} C_VEL
LIN {X 0,Y 474.581,Z 281.372,A -85,B 0,C 180,E1 -7262.688,E2 -7262.688} C_VEL
LIN {X 0,Y 474.611,Z 281.486,A -85,B 0,C 180,E1 -7264.074,E2 -7264.074} C_VEL
LIN {X 0,Y 477.763,Z 296.141,A -85,B 0,C 180,E1 -7266.441,E2 -7266.441} C_VEL
LIN {X 0,Y 476.854,Z 315.676,A -85,B 0,C 180,E1 -7269.289,E2 -7269.289} C_VEL
LIN {X 0,Y 476.027,Z 335.682,A -85,B 0,C 180,E1 -7272.164,E2 -7272.164} C_VEL
LIN {X 0,Y 475.687,Z 345.041,A -85,B 0,C 180,E1 -7273.499,E2 -7273.499} C_VEL
LIN {X 0,Y 477.563,Z 359.698,A -85,B 0,C 180,E1 -7273.795,E2 -7273.795} C_VEL
LIN {X 0,Y 476.829,Z 451.282,A -85,B 0,C 180,E1 -7275.247,E2 -7275.247} C_VEL
LIN {X 0,Y 476.637,Z 460.982,A -85,B 0,C 180,E1 -7275.486,E2 -7275.486} C_VEL
LIN {X 0,Y 476.321,Z 471.464,A -85,B 0,C 180,E1 -7275.858,E2 -7275.858} C_VEL
LIN {X 0,Y 476.016,Z 481.599,A -85,B 0,C 180,E1 -7276.339,E2 -7276.339} C_VEL
LIN {X 0,Y 475.634,Z 492.131,A -85,B 0,C 180,E1 -7276.981,E2 -7276.981} C_VEL
LIN {X 0,Y 475.338,Z 501.878,A -85,B 0,C 180,E1 -7277.72,E2 -7277.72} C_VEL
LIN {X 0,Y 475.065,Z 509.201,A -85,B 0,C 180,E1 -7278.374,E2 -7278.374} C_VEL
LIN {X 0,Y 474.679,Z 518.145,A -85,B 0,C 180,E1 -7279.337,E2 -7279.337} C_VEL
LIN {X 0,Y 474.382,Z 526.347,A -85,B 0,C 180,E1 -7280.408,E2 -7280.408} C_VEL
LIN {X 0,Y 474.139,Z 533.158,A -85,B 0,C 180,E1 -7281.478,E2 -7281.478} C_VEL
LIN {X 0,Y 473.996,Z 537.852,A -85,B 0,C 180,E1 -7282.334,E2 -7282.334} C_VEL
LIN {X 0,Y 473.878,Z 543.282,A -85,B 0,C 180,E1 -7283.543,E2 -7283.543} C_VEL
LIN {X 0,Y 473.833,Z 548.023,A -85,B 0,C 180,E1 -7284.897,E2 -7284.897} C_VEL
LIN {X 0,Y 473.757,Z 550.354,A -85,B 0,C 180,E1 -7285.748,E2 -7285.748} C_VEL
LIN {X 0,Y 473.779,Z 553.752,A -85,B 0,C 180,E1 -7287.451,E2 -7287.451} C_VEL
